// TwinCAT 3 PLC project Fraktal_Core
// Title: Fraktal_Core
// Company: fraktal-automation
// Author: fraktal-automation
// ProjectVersion: 0.1.0.5
// Description: Fraktal Core framework library: contracts, base classes (CM/EM/Unit), PermIntlk, profiler, connector base, recipe provider (Core 2.2).
// ProgramVersion: 3.1.4026.24
// libraries:
//   Tc2_Standard, * (Beckhoff Automation GmbH)
//   Tc2_EtherCAT, * (Beckhoff Automation GmbH)
//   Tc2_System, * (Beckhoff Automation GmbH)
//   Tc2_Utilities, * (Beckhoff Automation GmbH)
//   Tc3_Module, * (Beckhoff Automation GmbH)
// project tree:
//   BaseClasses/ FB_AccessManager.TcPOU, FB_AlarmLog.TcPOU, FB_AsciiDeviceCM.TcPOU, FB_ConfigPager.TcPOU, FB_ModuleBase.TcPOU, FB_ControlModuleBase.TcPOU (not stored), FB_CycleProfiler.TcPOU, FB_CompositeModuleBase.TcPOU, FB_EquipmentModuleBase.TcPOU (not stored), FB_SequenceBase.TcPOU (not stored), FB_UnitBase.TcPOU
//   Connectivity/ F_AppendTopologyConfig.TcPOU, FB_DeviceConnectorBase.TcPOU, FB_EcBusHealth.TcPOU, FB_EcFieldbusScanner.TcPOU (not stored), FB_IoTopologyPublisher.TcPOU, FB_LocalAccessProvider.TcPOU (not stored), FB_LocalPartCarrier.TcPOU (not stored), FB_LocalRecipeProvider.TcPOU (not stored), FB_LocalStationConfig.TcPOU, FB_SimByteChannel.TcPOU (not stored), FB_TcpChannelTc3.TcPOU (not stored)
//   DUTs/ E_AccessLevel.TcDUT (not stored), E_AlarmState.TcDUT (not stored), E_ByteChannelState.TcDUT (not stored), E_CarrierKind.TcDUT (not stored), E_Category.TcDUT (not stored), E_ChannelDir.TcDUT (not stored), E_ChannelKind.TcDUT (not stored), E_ExecState.TcDUT (not stored), E_FieldbusLossReaction.TcDUT (not stored), E_GatedAction.TcDUT (not stored), E_HbResult.TcDUT (not stored), E_LinkReaction.TcDUT (not stored), E_MachineState.TcDUT (not stored), E_Mode.TcDUT (not stored), E_ModeSwitchShield.TcDUT (not stored), E_PowerGroupKind.TcDUT (not stored), E_PowerState.TcDUT (not stored), E_SafetyDeviceKind.TcDUT (not stored), E_SafetyState.TcDUT (not stored), E_ModeSwitchStyle.TcDUT (not stored), E_ModuleType.TcDUT (not stored), E_NodeState.TcDUT (not stored), E_Reason.TcDUT (not stored), E_RecipeSource.TcDUT (not stored), E_ReleaseKind.TcDUT (not stored), E_ResetClass.TcDUT (not stored), E_RunStyle.TcDUT (not stored), E_Severity.TcDUT (not stored), E_StepResult.TcDUT (not stored), E_TimeClass.TcDUT (not stored), E_Verdict.TcDUT (not stored), ST_AccessPolicy.TcDUT (not stored), ST_AlarmEvent.TcDUT (not stored), ST_AlarmMeta.TcDUT (not stored), ST_BusNode.TcDUT (not stored), ST_CommandInfo.TcDUT (not stored), ST_CondRecord.TcDUT (not stored), ST_CycleProfile.TcDUT (not stored), ST_CycleSummary.TcDUT (not stored), ST_DecisionRequest.TcDUT (not stored), ST_Diagnostic.TcDUT (not stored), ST_FieldbusTopology.TcDUT (not stored), E_HmiRequestKind.TcDUT, ST_HmiRequest.TcDUT (not stored), ST_ConfigEntry.TcDUT, ST_ConfigPage.TcDUT, ST_HmiResponse.TcDUT (not stored), ST_IntlkCond.TcDUT (not stored), ST_IoChannel.TcDUT, ST_IoPointIdentity.TcDUT (not stored), ST_MeasRecord.TcDUT (not stored), ST_ModePolicy.TcDUT (not stored), ST_ModelField.TcDUT (not stored), ST_ModelId.TcDUT (not stored), ST_ModuleStatus.TcDUT (not stored), ST_ControlDomainStatus.TcDUT (not stored), ST_ControlPowerStatus.TcDUT (not stored), ST_PowerGroupStatus.TcDUT (not stored), ST_SafetyDeviceStatus.TcDUT (not stored), ST_SafetyStatus.TcDUT (not stored), ST_ModuleTiming.TcDUT (not stored), ST_Nameplate.TcDUT (not stored), ST_Oee.TcDUT (not stored), ST_OeeSample.TcDUT (not stored), ST_PartContext.TcDUT (not stored), ST_PartResult.TcDUT (not stored), ST_ReleaseReason.TcDUT (not stored), ST_ReleaseReport.TcDUT (not stored), ST_StepRecord.TcDUT, ST_StepTiming.TcDUT, ST_TimingRow.TcDUT (not stored), ST_UserRecord.TcDUT (not stored), ST_TcpVisionParCfg.TcDUT (not stored), ST_TcpVisionParCmd.TcDUT (not stored), ST_TcpVisionOutCmd.TcDUT (not stored), ST_TcpVisionOutImm.TcDUT (not stored), ST_TcpCodeReaderParCfg.TcDUT (not stored), ST_TcpCodeReaderParCmd.TcDUT (not stored), ST_TcpCodeReaderOutCmd.TcDUT (not stored), ST_TcpCodeReaderOutImm.TcDUT (not stored)
//   DeviceCMs/ FB_TcpCodeReaderCM.TcPOU, FB_TcpVisionCM.TcPOU (not stored)
//   Interfaces/ I_AccessProvider.TcIO (not stored), I_ByteChannel.TcIO (not stored), I_ControlModule.TcIO (not stored), I_DeviceConnector.TcIO (not stored), I_EquipmentModule.TcIO (not stored), I_EventSink.TcIO (not stored), I_FieldbusScanner.TcIO (not stored), I_ConfigSource.TcIO, I_Module.TcIO (not stored), I_PartCarrier.TcIO (not stored), I_SequenceHost.TcIO, I_RecipeProvider.TcIO (not stored), I_StationConfig.TcIO (not stored), I_Unit.TcIO (not stored), I_VerdictProvider.TcIO (not stored)
//   Params/ PL_Fraktal.TcGVL (not stored), PL_FraktalCompat.TcGVL (not stored), PL_TcpDevReasons.TcGVL (not stored)
//   PermIntlk/ FB_PermIntlk.TcPOU (not stored)
//   Platform/ F_Now.TcPOU (not stored), F_TimingUpdate.TcPOU (not stored)
// real-time tasks:
//   TASK PlcTask: cycle T#10ms, priority 20, ADS port 350
// I/O:
//   DEVICE =000+S-A610-A1 (EtherCAT), AmsNetId 0.0.0.0.2.1
//     =000+S-K010 (EK1200) [EK1200-5000 EtherCAT Power supply (2A E-Bus)]
//       =000+S-K010B1 (EL1809) [EL1809 16Ch. Dig. Input 24V, 3ms]
//       =000+S-K010C1 (EL2809) [EL2809 16Ch. Dig. Output 24V, 0.5A]
//       =000+S-K010D1 (EL6001) [EL6001 Interface (RS232)]
//       =000+S-K010E (EL9011) [EL9011 End Terminal]

// ---- DUTs/E_HmiRequestKind.TcDUT
// Core §3.10/§14 — generic OPC UA request mailbox operation.
// Append-only: ordinal values are a transport contract with every HMI adapter.
{attribute 'qualified_only'}
TYPE E_HmiRequestKind :
(
    NONE             := 0,
    LOGIN            := 1,
    LOGOUT           := 2,
    SET_MODE         := 3,
    SET_MODEL        := 4,
    START            := 5,
    STOP             := 6,
    CONTROL_ON       := 7,
    CONTROL_OFF      := 8,
    OPERATOR_RESET   := 9,
    DECISION_ANSWER  := 10,
    MANUAL_COMMAND   := 11,
    SET_RUN_STYLE    := 12,
    STEP_REQUEST     := 13,
    SET_HOLD_RUN     := 14,
    RELEASE_START    := 15,
    RELEASE_MANUAL   := 16,
    RELEASE_ACTION   := 17,
    RESET_OEE        := 18,
    WRITE_CONFIG     := 19,
    SHELVE_ALARM     := 20,
    UNSHELVE_ALARM   := 21,
    FORCE_CHANNEL    := 22,
    QUERY_CONFIG     := 23    // §3.10.2 config-manifest page request (IntValue = page)
) DINT;
END_TYPE

// ---- DUTs/ST_ConfigEntry.TcDUT
// Core §3.10.2 — one configuration value served through the request mailbox
// instead of the cyclic OPC UA tree. Scope selects the owner ('' = the root
// Unit itself, a qualified dotted module identity for a child, '#Fieldbus' for
// the bus topology). Item is the value's browse fragment in the server's array
// naming (e.g. 'Catalog/Catalog[2]/Label') so a generic HMI can rebuild the
// exact published path it would otherwise have read.
TYPE ST_ConfigEntry :
STRUCT
    Scope     : STRING(255);
    Item      : STRING(255);
    ValueText : STRING(255);   // typed by the HMI from the Item vocabulary
END_STRUCT
END_TYPE

// ---- DUTs/ST_ConfigPage.TcDUT
// Core §3.10.2 — one bounded page of the configuration manifest, published in
// ST_HmiResponse. The HMI requests QUERY_CONFIG with IntValue = PageIndex and
// walks 0..PageCount-1; Revision lets it detect a changed manifest (activation,
// changeover, config write) and refetch.
TYPE ST_ConfigPage :
STRUCT
    Revision   : UDINT;
    PageIndex  : INT;
    PageCount  : INT;
    EntryCount : INT;
    Entries    : ARRAY[1..PL_Fraktal.MAX_CONFIG_PAGE] OF ST_ConfigEntry;
END_STRUCT
END_TYPE

// ---- DUTs/ST_IoChannel.TcDUT
// Core §10.5.1 — one fieldbus I/O channel (published for the topology view §3.13)
TYPE ST_IoChannel :
STRUCT
    // §3.10.2 — tag/wiring identity is activation-static: excluded from the
    // cyclic OPC UA tree and served via the config manifest. Live I/O state
    // (values, force, quality, fault) stays cyclically published.
    {attribute 'OPC.UA.DA' := '0'}
    Name       : STRING(80);
    {attribute 'OPC.UA.DA' := '0'}
    DescriptionKey : STRING(160); // project/standard localization key
    {attribute 'OPC.UA.DA' := '0'}
    Address    : STRING(80);    // physical locator, e.g. EL1809 Ch5
    {attribute 'OPC.UA.DA' := '0'}
    Path       : STRING(255);   // unique channel path (force/audit identity)
    {attribute 'OPC.UA.DA' := '0'}
    ModulePath : STRING(255);   // owning module browse path for cross-navigation
    {attribute 'OPC.UA.DA' := '0'}
    Dir        : E_ChannelDir;
    {attribute 'OPC.UA.DA' := '0'}
    Kind       : E_ChannelKind;
    BoolValue  : BOOL;          // digital
    AnalogValue: REAL;          // analog (scaled)
    {attribute 'OPC.UA.DA' := '0'}
    Unit       : STRING(16);
    Forced     : BOOL;
    Quality    : BOOL;          // TRUE = good
    FaultActive: BOOL;          // a module diagnostic implicates this exact channel
    Diagnostic : STRING(255);   // localization key; Name remains the exact I/O tag
END_STRUCT
END_TYPE

// ---- DUTs/ST_StepRecord.TcDUT
// Core §6.5 — what the stall walk reads
TYPE ST_StepRecord :
STRUCT
    StepNo        : INT;
    StepName      : STRING(120);   // localization key
    AwaitingLabel : STRING(120);   // e.g. 'ClampStation.CLAMP' ('' if none)
    TimeClass     : E_TimeClass;   // Core §8.11.4(f) — WORK unless a genuine wait
    ExpectedTime  : TIME;          // defaults from the awaited command's timeout
    Conds         : ARRAY[1..PL_Fraktal.MAX_STEP_CONDS] OF ST_CondRecord;
END_STRUCT
END_TYPE

// ---- DUTs/ST_StepTiming.TcDUT
// Core §8.11.4(b)/(f) — one step of a cycle profile (Gantt/waterfall row)
TYPE ST_StepTiming :
STRUCT
    StepNo   : INT;
    StepName : STRING(120);   // localization key
    TimeClass    : E_TimeClass;  // WORK unless the step declared a wait class (§8.11.4(f))
    Started  : DT;           // synchronized wall clock (Core §2.7) — aligns across stations
    Duration : TIME;         // monotonic-clock duration (TC3 §8.11)
    Expected : TIME;         // §8.11.4(c) — the step's declared guard, drawn vs actual (0 = none)
END_STRUCT
END_TYPE

// ---- Interfaces/I_ConfigSource.TcIO
// Core §3.10.2 — a module that contributes entries to the root Unit's
// configuration manifest (static data deliberately excluded from the cyclic
// OPC UA tree and served through the QUERY_CONFIG mailbox instead).
// FB_ModuleBase implements it once for the base-owned facets; composites
// recurse their children, so a new module type inherits participation and
// only overrides M_AppendConfig to add type-owned static data (rare).
INTERFACE I_ConfigSource EXTENDS __System.IQueryInterface

// Append this module's (and its children's) manifest entries to the pager.
// Deterministic order across calls — the walk order defines the paging.
METHOD M_AppendConfig : BOOL
VAR_INPUT
    Pager : REFERENCE TO FB_ConfigPager;
END_VAR
END_METHOD

END_INTERFACE

// ---- Interfaces/I_SequenceHost.TcIO
// Core §6.7/§6.8 — the bridge from a separately-compiled sequence POU (SFC/ST/LD)
// to its owning module's protected framework services: step record, condition
// waits, run-style gate, part lifecycle, decisions, and completion/fault.
// FB_UnitBase implements it once; a sequence receives it at Setup. It carries
// framework plumbing ONLY — application decisions stay in the sequence's steps.
INTERFACE I_SequenceHost

// §6.11 publish a decision request
METHOD M_SequenceAskDecision
VAR_INPUT
    Req : ST_DecisionRequest;
END_VAR
END_METHOD

// §6.9(b) named plain-condition wait
METHOD M_SequenceAwait : BOOL
VAR_INPUT
    Idx : INT;
    Label : STRING(120);
    Ok : BOOL;
END_VAR
END_METHOD

// §6.11 withdraw an open request
METHOD M_SequenceClearDecision
END_METHOD

// §6.1 one-shot sequence completion (finite chains)
METHOD M_SequenceComplete
END_METHOD

// §8.11.2 carrier-less fallback counter
METHOD M_SequenceCountGood
END_METHOD

// §8.11.1 cycle-complete marker; FALSE = stop granted (chain must not loop)
METHOD M_SequenceEndOfCycle : BOOL
END_METHOD

// §6.9 first-out fault from a step
METHOD M_SequenceFault
VAR_INPUT
    Reason : E_Reason;
    DescriptionKey : STRING(255);
END_VAR
END_METHOD

// §3.16.3 EVENT_PART_PROCESSED (write-result-first; counts by verdict §8.11.2)
METHOD M_SequencePartProcessed : BOOL
VAR_INPUT
    Verdict : E_Verdict;
    Reason : E_Reason;
END_VAR
END_METHOD

// §3.16.3 EVENT_PART_RECEIVED
METHOD M_SequencePartReceived : BOOL
END_METHOD

// §3.16.1 measured value
METHOD M_SequencePartRecord : BOOL
VAR_INPUT
    RecordName : STRING(64);
    Value : LREAL;
    Minimum : LREAL;
    Maximum : LREAL;
    Target : LREAL;
    EngUnit : STRING(16);
END_VAR
END_METHOD

// §3.16.3 EVENT_PART_PROCESSING_STARTED
METHOD M_SequencePartStarted
END_METHOD

// §6.5 step record (feeds the §6.9 walk and the §8.11.4 profiler)
METHOD M_SequenceSetStep
VAR_INPUT
    StepNo : INT;
    StepName : STRING(120);
    Awaits : I_Module;
    AwaitingLabel : STRING(120);
    TimeClass : E_TimeClass;
    ExpectedTime : TIME;
END_VAR
END_METHOD

// §3.4.2 run-style pacing gate
METHOD M_SequenceStepGate : BOOL
VAR_INPUT
    Steppable : BOOL;
END_VAR
END_METHOD

// §3.4/§8.11 — accept a pending Stop BETWEEN cycles: abandon the open cycle
// profile (no §8.11.1 cycle is counted for a wait-only fragment) and complete.
METHOD M_SequenceStopNow
END_METHOD

// §3.4 — TRUE while a Stop is requested and the sequence still runs. A chain
// polls this at its between-cycles wait so a stop need not ride out a phantom cycle.
METHOD M_SequenceStopPending : BOOL
END_METHOD

// §6.11 consume the answer once (0 = none yet)
METHOD M_SequenceTakeDecision : INT
END_METHOD

END_INTERFACE

// ---- BaseClasses/FB_AccessManager.TcPOU
// Core §7.7(c) — per-root session + enforcement. Login/logout is DATA-DRIVEN
// (§3.10(a')): the HMI writes ReqUser/ReqSecret and pulses ReqLogin/ReqLogout;
// the secret is cleared after every attempt. Policy default: fully open (§7.7(b)).
FUNCTION_BLOCK FB_AccessManager
VAR_INPUT
    ReqUser   : STRING(32);          // HMI-writable login request
    ReqSecret : STRING(32);          // cleared after each attempt (§7.7(c))
    ReqLogin  : BOOL;
    ReqLogout : BOOL;
END_VAR
VAR_OUTPUT
    CurrentUser  : STRING(32);
    CurrentLevel : E_AccessLevel;    // HMI greys controls from this; PLC re-checks
    LoginFailed  : BOOL;             // last attempt outcome (HMI feedback)
END_VAR
VAR PERSISTENT
    Policy : ST_AccessPolicy;        // §3.8a station config; edit gated by ACCESS_POLICY
END_VAR
VAR
    {attribute 'OPC.UA.DA' := '0'}
    _provider : I_AccessProvider;
    {attribute 'OPC.UA.DA' := '0'}
    _log      : POINTER TO FB_AlarmLog;
    _tIdle    : TON;
END_VAR

// event/session handling is in Cyclic (called by the owning Unit each scan)

METHOD Cyclic : BOOL
VAR
    lvl : E_AccessLevel;
    loginHandled : BOOL;
    logoutHandled : BOOL;
END_VAR
loginHandled := ReqLogin;
IF loginHandled THEN
    ReqLogin := FALSE;
    lvl := E_AccessLevel.NONE;
    IF _provider <> 0 THEN
        lvl := _provider.Authenticate(User := ReqUser, Secret := ReqSecret);
    END_IF
    ReqSecret := '';                                   // never retain the secret
    IF lvl > E_AccessLevel.NONE THEN
        CurrentUser := ReqUser;
        CurrentLevel := lvl;
        LoginFailed := FALSE;
        _M_Audit('std.audit.login', CurrentUser);
    ELSE
        LoginFailed := TRUE;
        _M_Audit('std.audit.loginFailed', ReqUser);
    END_IF
END_IF
logoutHandled := ReqLogout;
IF logoutHandled THEN
    ReqLogout := FALSE;
    IF CurrentLevel > E_AccessLevel.NONE THEN
        _M_Audit('std.audit.logout', CurrentUser);
        CurrentUser := '';
        CurrentLevel := E_AccessLevel.NONE;
    END_IF
END_IF
// idle auto-logout (§7.7(c)); any successful login rearms it
_tIdle(IN := (Policy.SessionTimeout > T#0S) AND (CurrentLevel > E_AccessLevel.NONE) AND NOT loginHandled,
       PT := Policy.SessionTimeout);
IF _tIdle.Q THEN
    _M_Audit('std.audit.autoLogout', CurrentUser);
    CurrentUser := '';
    CurrentLevel := E_AccessLevel.NONE;
END_IF
Cyclic := TRUE;
END_METHOD

// Startup/station-configuration seam; runtime HMI writes remain Unit-gated.
METHOD ConfigureRequired : BOOL
VAR_INPUT
    Gate : E_GatedAction;
    Level : E_AccessLevel;
END_VAR
IF (TO_INT(Gate) < 0) OR (TO_INT(Gate) > TO_INT(E_GatedAction.POWER_CONTROL)) THEN
    ConfigureRequired := FALSE;
ELSE
    Policy.Required[TO_INT(Gate)] := Level;
    ConfigureRequired := TRUE;
END_IF
END_METHOD

// ST-facing request seam. OPC UA clients continue to write the published request data.
METHOD RequestLogin : BOOL
VAR_INPUT
    User : STRING(32);
    Secret : STRING(32);
END_VAR
ReqUser := User;
ReqSecret := Secret;
ReqLogin := TRUE;
RequestLogin := TRUE;
END_METHOD

// ST-facing request seam; the cyclic edge handler performs the state change and audit.
METHOD RequestLogout : BOOL
ReqLogout := TRUE;
RequestLogout := TRUE;
END_METHOD

// pure check for UI/logic — no logging
METHOD Permits : BOOL
VAR_INPUT
    Gate : E_GatedAction;
END_VAR
Permits := TO_DINT(CurrentLevel) >= TO_DINT(Policy.Required[TO_INT(Gate)]);
END_METHOD

// gated-entry check: a DENIED attempt is audited as a MESSAGE event (§8.3/§7.7(c))
METHOD PermitsLogged : BOOL
VAR_INPUT
    Gate : E_GatedAction;
END_VAR
PermitsLogged := Permits(Gate := Gate);
IF NOT PermitsLogged THEN
    _M_Audit('std.audit.accessDenied', CurrentUser);
END_IF
END_METHOD

METHOD Setup : BOOL
VAR_INPUT
    Provider : I_AccessProvider;
    pAlarmLog : POINTER TO FB_AlarmLog;
END_VAR
IF Provider <> 0 THEN
    _provider := Provider;                  // Unit OnInit may attach only the audit log
END_IF
_log := pAlarmLog;
Setup := TRUE;
END_METHOD

// audit trail for free: come+gone MESSAGE lands in the §8.3 ring
METHOD PRIVATE _M_Audit
VAR_INPUT
    What : STRING(64);
    Who : STRING(32);
END_VAR
VAR
    auditSlot : INT;
    txt : STRING(255);
END_VAR
IF _log = 0 THEN
    RETURN;
END_IF
txt := CONCAT(What, ': ');
txt := CONCAT(txt, Who);
auditSlot := _log^.Raise(Reason := E_Reason.NONE, Text := txt,
                 Source := 'Access', Severity := E_Severity.LOW,
                 Category := E_Category.SYSTEM, ResetClass := E_ResetClass.AUTO_RESET);
IF auditSlot > 0 THEN
    _log^.Gone(Slot := auditSlot);                     // instant come+gone -> ring entry
END_IF
END_METHOD

END_FUNCTION_BLOCK

// ---- BaseClasses/FB_AlarmLog.TcPOU
// Core §8.3 — per-Unit alarm & event log: active list + closed ring, durations,
// AUTO/MANUAL reset classes, optional historian sink. Fixed-size, never allocates.
FUNCTION_BLOCK FB_AlarmLog
VAR_OUTPUT
    Active    : ARRAY[1..PL_Fraktal.MAX_ALARM_ACTIVE] OF ST_AlarmEvent;  // ACTIVE/WAIT_RESET
    NActive   : INT;
    Ring      : ARRAY[1..PL_Fraktal.MAX_ALARM_RING] OF ST_AlarmEvent;    // closed, newest at RingHead
    RingHead  : INT;
    Blocking  : BOOL;    // any MANUAL_RESET event ACTIVE/WAIT_RESET (§8.3(b))
    Truncated : BOOL;
    // §3.10.2 — rationalization records are static config; excluded from the
    // cyclic OPC UA tree (served via the manifest when an HMI needs them).
    {attribute 'OPC.UA.DA' := '0'}
    Meta      : ARRAY[1..PL_Fraktal.MAX_ALARM_META] OF ST_AlarmMeta;  // §8.9 rationalization
    {attribute 'OPC.UA.DA' := '0'}
    MetaCount : INT;
END_VAR
VAR
    {attribute 'OPC.UA.DA' := '0'}
    _sink    : I_EventSink;
    _comeMs  : ARRAY[1..PL_Fraktal.MAX_ALARM_ACTIVE] OF DWORD;   // monotonic (TC3 §8.11)
    _shelfMs : ARRAY[1..PL_Fraktal.MAX_ALARM_ACTIVE] OF UDINT;   // §8.10 countdown (0 = not shelved)
    _cycLast : TIME;                                             // Cyclic delta stamp
END_VAR

// event-driven; no cyclic body

// §8.3(c) — open a non-channel-specific event; returns slot (0 = full).
METHOD Raise : INT
VAR_INPUT
    Reason : E_Reason;
    Text : STRING(255);
    Source : STRING(255);
    Severity : E_Severity;
    Category : E_Category;
    ResetClass : E_ResetClass;
END_VAR
Raise := _M_Raise(Reason := Reason, Text := Text, Source := Source,
    IoTag := '', IoAddress := '', Severity := Severity, Category := Category,
    ResetClass := ResetClass);
END_METHOD

// §8.3(c) — open an event; returns its slot id (0 = table full -> Truncated)
METHOD PRIVATE _M_Raise : INT
VAR_INPUT
    Reason : E_Reason;
    Text : STRING(255);
    Source : STRING(255);
    IoTag : STRING(80);
    IoAddress : STRING(80);
    Severity : E_Severity;
    Category : E_Category;
    ResetClass : E_ResetClass;
END_VAR
VAR
    i, slot : INT;
END_VAR
slot := 0;
FOR i := 1 TO PL_Fraktal.MAX_ALARM_ACTIVE DO
    IF Active[i].State = E_AlarmState.CLOSED THEN
        slot := i;
        EXIT;
    END_IF
END_FOR
IF slot = 0 THEN
    Truncated := TRUE;
    _M_Raise := 0;
    RETURN;
END_IF
Active[slot].ReasonCode  := Reason;
Active[slot].Description := Text;
Active[slot].SourcePath  := Source;
Active[slot].IoTag       := IoTag;
Active[slot].IoAddress   := IoAddress;
Active[slot].Severity    := Severity;
Active[slot].Category    := Category;
Active[slot].ResetClass  := ResetClass;
Active[slot].State       := E_AlarmState.ACTIVE;
Active[slot].ComeAt      := F_Now();
Active[slot].GoneAt      := DT#1970-01-01-00:00:00;
Active[slot].ResetAt     := DT#1970-01-01-00:00:00;
Active[slot].Duration    := T#0S;
Active[slot].Shelved     := FALSE;
Active[slot].ShelvedUntil:= DT#1970-01-01-00:00:00;
_shelfMs[slot] := 0;
_comeMs[slot] := TIME_TO_DWORD(TIME());
NActive := NActive + 1;
_M_UpdateBlocking();
IF _sink <> 0 THEN
    _sink.OnEvent(Ev := Active[slot]);              // come notification (§8.3(d))
END_IF
_M_Raise := slot;
END_METHOD

// §8.3(c) — open an ERROR event straight from a first-out diagnostic (no re-authoring)
METHOD RaiseDiag : INT
VAR_INPUT
    D : ST_Diagnostic;
    ResetClass : E_ResetClass;
END_VAR
RaiseDiag := _M_Raise(Reason := D.ReasonCode, Text := D.Description,
                   Source := D.SourcePath, IoTag := D.IoTag, IoAddress := D.IoAddress,
                   Severity := D.Severity, Category := D.Category,
                   ResetClass := ResetClass);
END_METHOD

// §8.3(b) — condition re-established: AUTO_RESET closes with Duration;
// MANUAL_RESET stays blocking in WAIT_RESET until OperatorReset.
METHOD Gone : BOOL
VAR_INPUT
    Slot : INT;
END_VAR
Gone := FALSE;
IF (Slot < 1) OR (Slot > PL_Fraktal.MAX_ALARM_ACTIVE) THEN
    RETURN;
END_IF
IF Active[Slot].State <> E_AlarmState.ACTIVE THEN
    RETURN;
END_IF
Active[Slot].GoneAt   := F_Now();
Active[Slot].Duration := DWORD_TO_TIME(TIME_TO_DWORD(TIME()) - _comeMs[Slot]);   // wrap-safe
IF Active[Slot].ResetClass = E_ResetClass.AUTO_RESET THEN
    _M_Close(Slot);
ELSE
    Active[Slot].State := E_AlarmState.WAIT_RESET;   // still blocking (§8.3(b))
END_IF
Gone := TRUE;
END_METHOD

// §8.3(b) — deliberate, release-gated operator action (§7.6/§14): closes
// MANUAL_RESET events whose condition is gone. NEVER self-invoked (§9.3 principle).
METHOD OperatorReset : BOOL
VAR
    i : INT;
END_VAR
OperatorReset := FALSE;
FOR i := 1 TO PL_Fraktal.MAX_ALARM_ACTIVE DO
    IF Active[i].State = E_AlarmState.WAIT_RESET THEN
        Active[i].ResetAt := F_Now();
        _M_Close(i);
        OperatorReset := TRUE;
    END_IF
END_FOR
END_METHOD

METHOD SetSink : BOOL
VAR_INPUT
    Sink : I_EventSink;
END_VAR
_sink := Sink;
SetSink := TRUE;
END_METHOD

METHOD PRIVATE _M_Close
VAR_INPUT
    Slot : INT;
END_VAR
Active[Slot].State := E_AlarmState.CLOSED;
RingHead := (RingHead MOD PL_Fraktal.MAX_ALARM_RING) + 1;
Ring[RingHead] := Active[Slot];
Ring[RingHead].State := E_AlarmState.CLOSED;
NActive := NActive - 1;
_M_UpdateBlocking();
IF _sink <> 0 THEN
    _sink.OnEvent(Ev := Ring[RingHead]);            // close notification with Duration (§8.3(d))
END_IF
END_METHOD

METHOD PRIVATE _M_UpdateBlocking
VAR
    i : INT;
    b : BOOL;
END_VAR
b := FALSE;
FOR i := 1 TO PL_Fraktal.MAX_ALARM_ACTIVE DO
    IF (Active[i].ResetClass = E_ResetClass.MANUAL_RESET)
    AND (Active[i].State <> E_AlarmState.CLOSED) THEN
        b := TRUE;
        EXIT;
    END_IF
END_FOR
Blocking := b;
END_METHOD

// §8.9 — register/update the rationalization record for a ReasonCode (idempotent).
// Modules/Units call at Setup. No record => the reason is NOT shelvable (§8.10).
METHOD RegisterMeta : BOOL
VAR_INPUT
    Reason         : E_Reason;
    OperatorAction : STRING(255);
    Consequence    : STRING(255);
    Shelvable      : BOOL;
END_VAR
VAR
    i : INT;
END_VAR
FOR i := 1 TO MetaCount DO
    IF Meta[i].ReasonCode = Reason THEN
        Meta[i].OperatorAction := OperatorAction;
        Meta[i].Consequence := Consequence;
        Meta[i].Shelvable := Shelvable;
        RegisterMeta := TRUE;
        RETURN;
    END_IF
END_FOR
IF MetaCount >= PL_Fraktal.MAX_ALARM_META THEN
    RegisterMeta := FALSE;
    RETURN;
END_IF
MetaCount := MetaCount + 1;
Meta[MetaCount].ReasonCode := Reason;
Meta[MetaCount].OperatorAction := OperatorAction;
Meta[MetaCount].Consequence := Consequence;
Meta[MetaCount].Shelvable := Shelvable;
RegisterMeta := TRUE;
END_METHOD

// §8.10 — may this active slot be shelved? SAFETY never; no meta record => no.
METHOD PROTECTED _M_Shelvable : BOOL
VAR_INPUT
    Slot : INT;
END_VAR
VAR
    i : INT;
END_VAR
_M_Shelvable := FALSE;
IF Slot < 1 OR Slot > PL_Fraktal.MAX_ALARM_ACTIVE THEN
    RETURN;
END_IF
IF Active[Slot].State = E_AlarmState.CLOSED THEN
    RETURN;
END_IF
IF Active[Slot].Category = E_Category.SAFETY THEN
    RETURN;                              // §8.10: safety never shelvable
END_IF
FOR i := 1 TO MetaCount DO
    IF Meta[i].ReasonCode = Active[Slot].ReasonCode THEN
        _M_Shelvable := Meta[i].Shelvable;
        RETURN;
    END_IF
END_FOR
// no rationalization record => not shelvable (rationalize first, §8.10)
END_METHOD

// §8.10 — suppress ANNUNCIATION of an active alarm for DurationS seconds (capped).
// Control is untouched: Blocking, interlocks, release reports all still see it.
// Caller has already checked §7.7 ALARM_SHELVE; the shelf itself is logged here.
METHOD Shelve : BOOL
VAR_INPUT
    Slot      : INT;
    DurationS : UDINT;
END_VAR
VAR
    auditSlot : INT;
END_VAR
IF NOT _M_Shelvable(Slot := Slot) THEN
    Shelve := FALSE;
    RETURN;
END_IF
IF DurationS = 0 THEN
    Shelve := FALSE;                              // every shelf is time-bounded
    RETURN;
END_IF
IF DurationS > PL_Fraktal.MAX_SHELF_S THEN
    DurationS := PL_Fraktal.MAX_SHELF_S;         // §8.10 time-bounded
END_IF
Active[Slot].Shelved := TRUE;
Active[Slot].ShelvedUntil := DWORD_TO_DT(DT_TO_DWORD(F_Now()) + DurationS);
_shelfMs[Slot] := DurationS * 1000;
auditSlot := Raise(Reason := E_Reason.NONE,
    Text := 'std.audit.alarmShelved', Source := Active[Slot].SourcePath,
    Severity := E_Severity.LOW, Category := E_Category.SYSTEM, ResetClass := E_ResetClass.AUTO_RESET);
IF auditSlot > 0 THEN Gone(Slot := auditSlot); END_IF
Shelve := TRUE;
END_METHOD

// §8.10 — restore annunciation (operator or auto-expiry). Logged.
METHOD Unshelve : BOOL
VAR_INPUT
    Slot : INT;
END_VAR
VAR
    auditSlot : INT;
END_VAR
IF Slot < 1 OR Slot > PL_Fraktal.MAX_ALARM_ACTIVE THEN
    Unshelve := FALSE;
    RETURN;
END_IF
IF NOT Active[Slot].Shelved THEN
    Unshelve := FALSE;
    RETURN;
END_IF
Active[Slot].Shelved := FALSE;
_shelfMs[Slot] := 0;
auditSlot := Raise(Reason := E_Reason.NONE,
    Text := 'std.audit.alarmUnshelved', Source := Active[Slot].SourcePath,
    Severity := E_Severity.LOW, Category := E_Category.SYSTEM, ResetClass := E_ResetClass.AUTO_RESET);
IF auditSlot > 0 THEN Gone(Slot := auditSlot); END_IF
Unshelve := TRUE;
END_METHOD

// §8.10 — auto-unshelve countdown (owning Unit ticks this each scan).
METHOD Cyclic : BOOL
VAR
    currentTime : TIME;
    deltaMs     : UDINT;
    i   : INT;
END_VAR
currentTime := TIME();                 // monotonic duration clock
IF _cycLast = T#0S THEN
    _cycLast := currentTime;
    Cyclic := TRUE;
    RETURN;
END_IF
deltaMs := TIME_TO_UDINT(currentTime) - TIME_TO_UDINT(_cycLast);
_cycLast := currentTime;
FOR i := 1 TO PL_Fraktal.MAX_ALARM_ACTIVE DO
    IF Active[i].Shelved AND _shelfMs[i] > 0 THEN
        IF _shelfMs[i] > deltaMs THEN
            _shelfMs[i] := _shelfMs[i] - deltaMs;
        ELSE
            _shelfMs[i] := 0;
            Unshelve(Slot := i);                 // §8.10 auto-expire (logged by Unshelve)
        END_IF
    END_IF
END_FOR
Cyclic := TRUE;
END_METHOD

END_FUNCTION_BLOCK

// ---- BaseClasses/FB_AsciiDeviceCM.TcPOU
// Core §3.15.1a — CM base for ASCII request/response devices over I_ByteChannel
// (vision sensors, code readers, gauges). One-outstanding-request state machine:
// SendRequest -> await terminated response -> _M_OnResponse hook; silence -> fault
// 10402. Written ONCE against the neutral seam: porting = swap the channel (O4/O8).
// Reconnect: bounded retry via the channel; link state published for Annex D facet.
FUNCTION_BLOCK ABSTRACT FB_AsciiDeviceCM EXTENDS FB_ControlModuleBase
VAR
    Host        : STRING(80);          // §3.8 config (per deployment)
    Port        : UINT;
    Terminator  : STRING(2) := '$R';   // CR default; device profile may override
    RespTimeout : TIME := T#2S;
    LinkState   : E_ByteChannelState;  // published (Annex D link facet)
    LastResponse: STRING(255);         // published (diagnosis)
END_VAR
VAR
    {attribute 'OPC.UA.DA' := '0'}
    _chan     : I_ByteChannel;
    _rx       : STRING(255);
    _pending  : BOOL;                  // one outstanding request
    _tResp    : TON;
    _tRetry   : TON;
    _retryMs  : TIME := T#500MS;       // bounded backoff (doubles to 10s)
    _openTried : BOOL;                 // backoff spaces RE-tries; the first Open is immediate
END_VAR

;  // driven via Cyclic (base) -> OnCyclic below

// wire the transport + endpoint. Call from the profile's Setup after _M_SetName.
METHOD SetupDevice : BOOL
VAR_INPUT
    Chan : I_ByteChannel;
    DevHost : STRING(80);
    DevPort : UINT;
END_VAR
IF Chan = 0 OR DevHost = '' THEN
    _M_FaultN(PL_TcpDevReasons.DEV_CFG_INVALID, 'std.error.deviceConnectionNotConfigured');
    SetupDevice := FALSE;
    RETURN;
END_IF
_chan := Chan;
Host := DevHost;
Port := DevPort;
SetupDevice := TRUE;
END_METHOD

// channel management + RX framing. Profiles override _M_OnResponse, not this.
METHOD PROTECTED OnCyclic : DINT
VAR
    pos : INT;
    resp : STRING(255);
END_VAR
OnCyclic := SUPER^.OnCyclic();
IF _chan = 0 THEN
    RETURN;
END_IF
_chan.Tick();
LinkState := _chan.State();
CASE LinkState OF
    E_ByteChannelState.CLOSED:
        IF NOT _openTried THEN
            _openTried := TRUE;                    // first sight of CLOSED: connect NOW
            _chan.Open(Host := Host, Port := Port);
            LinkState := _chan.State();            // a synchronous transport is OPEN this scan
        ELSE
            _tRetry(IN := TRUE, PT := _retryMs);   // failed before: bounded backoff (§3.15.2 spirit)
            IF _tRetry.Q THEN
                _tRetry(IN := FALSE);
                _chan.Open(Host := Host, Port := Port);
                LinkState := _chan.State();
                IF _retryMs < T#10S THEN
                    _retryMs := _retryMs * 2;
                END_IF
            END_IF
        END_IF
    E_ByteChannelState.OPEN:
        _openTried := FALSE;
        _retryMs := T#500MS;
        _chan.Poll(Buffer := _rx);
        pos := FIND(_rx, Terminator);
        IF pos > 0 THEN
            resp := LEFT(_rx, pos - 1);
            _rx := DELETE(_rx, pos + LEN(Terminator) - 1, 1);
            _pending := FALSE;
            _tResp(IN := FALSE);
            LastResponse := resp;
            _M_OnResponse(Response := resp);
        ELSIF LEN(_rx) >= 250 THEN
            _rx := '';
            _M_FaultN(PL_TcpDevReasons.DEV_RX_OVERFLOW, 'std.error.deviceResponseOverflow');
        END_IF
    E_ByteChannelState.FAULT:
        IF _pending THEN
            _pending := FALSE;
            _tResp(IN := FALSE);
        END_IF
        _M_FaultN(PL_TcpDevReasons.DEV_CHANNEL_FAULT, 'std.error.transportChannelFault');
        _chan.Close();
ELSE
    _M_FaultN(PL_TcpDevReasons.DEV_CHANNEL_FAULT, 'std.error.byteChannelStateInvalid');
    _chan.Close();
END_CASE
// response timeout watch
_tResp(IN := _pending, PT := RespTimeout);
IF _tResp.Q THEN
    _pending := FALSE;
    _tResp(IN := FALSE);
    _M_FaultN(PL_TcpDevReasons.DEV_RESP_TIMEOUT, 'std.error.deviceResponseTimeout');
END_IF
END_METHOD

// issue one request (terminator appended). FALSE if not connected or one pending.
METHOD SendRequest : BOOL
VAR_INPUT
    Text : STRING(250);
END_VAR
// live channel state: the cached LinkState is one scan old and would reject a
// request issued in the same scan the transport opened.
IF _chan = 0 OR (_chan.State() <> E_ByteChannelState.OPEN) THEN
    _M_FaultN(PL_TcpDevReasons.DEV_NOT_CONNECTED, 'std.error.deviceNotConnected');
    SendRequest := FALSE;
    RETURN;
END_IF
IF _pending THEN
    SendRequest := FALSE;              // one-outstanding-request contract
    RETURN;
END_IF
_pending := _chan.Send(Text := CONCAT(Text, Terminator));
SendRequest := _pending;
END_METHOD

// profile hook: parse one terminated response. Raise DEV_PROTOCOL on garbage.
METHOD PROTECTED _M_OnResponse
VAR_INPUT
    Response : STRING(255);
END_VAR
;
END_METHOD

END_FUNCTION_BLOCK

// ---- BaseClasses/FB_ConfigPager.TcPOU
// Core §3.10.2 — windowed writer for the configuration manifest. QUERY_CONFIG
// re-walks the whole export enumeration each request; the pager counts every
// appended entry and stores only the requested page window into the published
// ST_ConfigPage, so no full manifest buffer ever exists in PLC memory and the
// walk order alone defines the paging. Exporters call M_Append*/ignore paging.
FUNCTION_BLOCK FB_ConfigPager
VAR
    {attribute 'OPC.UA.DA' := '0'}
    _pTarget : POINTER TO ST_ConfigPage;
    _cursor  : DINT;   // entries appended so far in this walk
    _first   : DINT;   // first cursor index stored in the window (0-based)
END_VAR

; // stateless between requests — driven entirely by M_Setup/M_Append/M_Finish

// Begin one QUERY_CONFIG walk targeting the published page window.
METHOD M_Setup : BOOL
VAR_INPUT
    Target    : POINTER TO ST_ConfigPage;
    PageIndex : INT;
    Revision  : UDINT;
END_VAR
M_Setup := FALSE;
IF Target = 0 THEN
    RETURN;
END_IF
_pTarget := Target;
_cursor := 0;
IF PageIndex < 0 THEN
    _first := 0;
ELSE
    _first := TO_DINT(PageIndex) * TO_DINT(PL_Fraktal.MAX_CONFIG_PAGE);
END_IF
_pTarget^.Revision := Revision;
_pTarget^.PageIndex := SEL(PageIndex < 0, PageIndex, 0);
_pTarget^.PageCount := 0;
_pTarget^.EntryCount := 0;
M_Setup := TRUE;
END_METHOD

// Append one manifest entry; stored only when it falls inside the page window.
// Always returns TRUE so exporters can chain without branching.
METHOD M_Append : BOOL
VAR_INPUT
    Scope     : STRING(255);
    Item      : STRING(255);
    ValueText : STRING(255);
END_VAR
VAR
    slot : DINT;
END_VAR
M_Append := TRUE;
IF _pTarget = 0 THEN
    RETURN;
END_IF
slot := _cursor - _first;   // window-relative 0-based position
_cursor := _cursor + 1;
IF (slot < 0) OR (slot >= TO_DINT(PL_Fraktal.MAX_CONFIG_PAGE)) THEN
    RETURN;                 // outside the requested window — counted, not stored
END_IF
_pTarget^.Entries[TO_INT(slot) + 1].Scope := Scope;
_pTarget^.Entries[TO_INT(slot) + 1].Item := Item;
_pTarget^.Entries[TO_INT(slot) + 1].ValueText := ValueText;
_pTarget^.EntryCount := TO_INT(slot) + 1;
END_METHOD

METHOD M_AppendNumber : BOOL
VAR_INPUT
    Scope  : STRING(255);
    Item   : STRING(255);
    Number : DINT;
END_VAR
M_AppendNumber := M_Append(Scope := Scope, Item := Item,
    ValueText := TO_STRING(Number));
END_METHOD

// Close the walk: publish the total page count for the HMI's fetch loop.
METHOD M_Finish : BOOL
M_Finish := FALSE;
IF _pTarget = 0 THEN
    RETURN;
END_IF
_pTarget^.PageCount := TO_INT(
    (_cursor + TO_DINT(PL_Fraktal.MAX_CONFIG_PAGE) - 1)
    / TO_DINT(PL_Fraktal.MAX_CONFIG_PAGE));
M_Finish := TRUE;
END_METHOD

END_FUNCTION_BLOCK

// ---- BaseClasses/FB_ModuleBase.TcPOU
// Core §2.2 / §6.1 — the PLCopen lifecycle written ONCE (template method).
// A concrete type EXTENDS this base, declares its Command/HAL/ParCfg members, and
// overrides only _M_Dispatch (+ optionally hooks and recipe transaction methods).
// Edge handling, ExecState mapping, Execute-drop reset, ErrorID publication, and
// abort routing are inherited. Conformance rows T1/T4 (Core §5.7) are satisfied here
// and proven once in FB_Base_Tests.
FUNCTION_BLOCK ABSTRACT FB_ModuleBase IMPLEMENTS I_Module, I_ConfigSource
VAR_INPUT
    Execute : BOOL;    // rising edge starts the command (Core §6.1)
    Abort   : BOOL;    // requests a controlled abort
END_VAR
VAR_OUTPUT
    Busy    : BOOL;
    Done    : BOOL;
    Error   : BOOL;
    Aborted : BOOL;
    ErrorID : DWORD;   // = TO_DWORD(first-out ReasonCode), Core §8.8
END_VAR
VAR_OUTPUT
    Status : ST_ModuleStatus;   // Core §3.10(a')/§6.9(a) — the OPC UA data mirror
    Timing : ST_ModuleTiming;   // Core §8.11.4(a) — per-command timing, captured here once
    // §3.10.2 — static facets stay OFF the cyclic OPC UA tree and are served
    // through the QUERY_CONFIG manifest instead (M_AppendConfig).
    {attribute 'OPC.UA.DA' := '0'}
    Nameplate   : ST_Nameplate;  // §3.10.1 asset identity (set at Setup; empty = none)
    {attribute 'OPC.UA.DA' := '0'}
    Catalog     : ARRAY[1..PL_Fraktal.MAX_CMD_CATALOG] OF ST_CommandInfo;  // §7.6.1 published command list
    {attribute 'OPC.UA.DA' := '0'}
    CatalogCount: INT;
    Safety       : ST_SafetyStatus;       // §9 optional read-only safety facet (Present=FALSE if absent)
    ControlPower : ST_ControlPowerStatus; // §9 optional control/power facet
END_VAR
VAR
    _name  : STRING(80);
    _exec  : E_ExecState := E_ExecState.READY;
    _step  : INT;
    _diag  : ST_Diagnostic;
    _rTrig : R_TRIG;
    _abortErrTrig : R_TRIG;
    _initialized : BOOL;
    _prevExec   : E_ExecState;
    _manualCmd  : DINT;          // §7.6.1 pending manual command value (0 = none)
    _manualReq  : BOOL;
    _manualActive : BOOL;        // one-shot manual request owns Execute until terminal state
    _cmdArmed   : BOOL;          // terminal state came from a command; gates the §6.1 reset
    _cmdId      : DINT;          // set by _M_TagCommand (one line per type, §8.11.4(a))
    _cmdLabel   : STRING(120);
    _tCmdStart  : DWORD;         // monotonic ms at command start (TC3 §8.11)
END_VAR

// FB body just runs the lifecycle; parents may call the instance or Cyclic() (I_Module)
Cyclic();

// Core §6.1 — edge -> hooks -> dispatch -> map -> Execute-drop reset
METHOD Cyclic : BOOL
VAR
    commandStarted : BOOL;
END_VAR
commandStarted := FALSE;
// Execute-drop reset (Core §6.1): a COMMAND-produced terminal state published in
// an earlier scan plus Execute low resets to READY BEFORE this scan's mapping, so
// the outputs go idle in the same call. A completion later this scan still maps
// its one-cycle DONE/ERROR/ABORTED pulse first (PLCopen). Faults raised OUTSIDE a
// command (recipe/config at Setup, cyclic condition monitors) latch (§3.8/§8.3):
// Execute was never high, so the handshake reset does not consume them.
IF (NOT Execute) AND _cmdArmed
AND ((_exec = E_ExecState.DONE) OR (_exec = E_ExecState.ERROR) OR (_exec = E_ExecState.ABORTED)) THEN
    _exec := E_ExecState.READY;
    _cmdArmed := FALSE;
END_IF

_rTrig(CLK := Execute);
// A fresh command edge may also RETRY from a latched non-command fault: the edge
// clears the diagnostic and re-runs validation, which re-faults if the cause remains.
IF _rTrig.Q AND ((_exec = E_ExecState.READY)
    OR ((_exec = E_ExecState.ERROR) AND NOT _cmdArmed)) THEN
    _exec := E_ExecState.BUSY;      // ParCmd of the concrete type is latched on this edge
    _cmdArmed := TRUE;
    _step := 10;
    _M_ClearDiag();
    _tCmdStart := TIME_TO_DWORD(TIME());          // §8.11.4(a) command-timing start
    commandStarted := TRUE;
END_IF

IF NOT _initialized THEN
    _initialized := TRUE;
    OnInit();                        // Core §3.14 one-shot for every module tier
END_IF
IF commandStarted THEN
    OnCommandStart();                // one-shot after init, before cyclic/dispatch
END_IF
OnCyclic();                          // Core §3.14 hook: background management, no outputs

IF Abort AND (_exec = E_ExecState.BUSY) THEN
    OnAbort();                       // Core §3.14 hook: device-safe abort action
END_IF
_abortErrTrig(CLK := Abort AND (_exec = E_ExecState.ERROR));
IF _abortErrTrig.Q THEN
    OnAbortInError();                // distinct recovery hook; ERROR remains latched
END_IF

IF _exec = E_ExecState.BUSY THEN
    _M_Dispatch();                   // the ONLY thing a type must write (Core §2.2)
END_IF

// §8.11.4(a) — close the command's timing row on leaving BUSY (DONE/ERROR/ABORTED)
IF (_prevExec = E_ExecState.BUSY) AND (_exec <> E_ExecState.BUSY) THEN
    _M_RecordCmdTiming(TIME_TO_DWORD(TIME()) - _tCmdStart);   // wrap-safe diff (TC3 §8.11)
END_IF
_prevExec := _exec;

Busy    := (_exec = E_ExecState.BUSY);
Done    := (_exec = E_ExecState.DONE);
Error   := (_exec = E_ExecState.ERROR);
Aborted := (_exec = E_ExecState.ABORTED);
ErrorID := TO_DWORD(_diag.ReasonCode);

// §6.9(a)/§3.10(a') — refresh the data mirror: properties are invisible to the
// OPC UA namespace, so everything the HMI binds is published here as DATA
Status.ModuleType  := ModuleType;
Status.State       := _exec;
Status.FaultActive := (_exec = E_ExecState.ERROR);
Status.Diagnostic  := _diag;
_M_PublishStatus();              // tier-specific overlay after the common mirror is final

// A manual command is a one-shot use of the same PLCopen lifecycle. Keep the
// terminal state visible for this scan, then drop Execute for next-scan reset.
IF _manualActive AND ((_exec = E_ExecState.DONE) OR (_exec = E_ExecState.ERROR) OR (_exec = E_ExecState.ABORTED)) THEN
    Execute := FALSE;
    _manualActive := FALSE;
END_IF
Cyclic := TRUE;
END_METHOD

// Core §8.2/§6.9 — this node's first-out (composites override via rollup in the EM base)
METHOD GetFaultSummary : ST_Diagnostic
GetFaultSummary := _diag;
END_METHOD

// Core §3.14 hook — optional override: device-safe abort action.
// Override contract (Core §3.14.2): call SUPER^.OnAbort() FIRST and keep its return.
METHOD PROTECTED OnAbort : DINT
_exec := E_ExecState.ABORTED;
_step := 0;
OnAbort := 0;
END_METHOD

// Core §3.14 — optional error-state abort/recovery action. ERROR remains latched
// until Execute drops. Overrides call SUPER^.OnAbortInError() first.
METHOD PROTECTED OnAbortInError : DINT
OnAbortInError := 0;
END_METHOD

// Core §3.14 — first operational scan, after Setup/recipe load.
// Overrides call SUPER^.OnInit() first and propagate its return.
METHOD PROTECTED OnInit : DINT
OnInit := 0;
END_METHOD

// Core §3.14 hook — optional override: per-scan background management (idempotent,
// no direct outputs). Override contract: call SUPER^.OnCyclic() FIRST, keep return.
METHOD PROTECTED OnCyclic : DINT
OnCyclic := 0;
END_METHOD

// Core §3.14 hook — one-shot on each accepted Execute rising edge, after OnInit
// and before OnCyclic/_M_Dispatch. Overrides call SUPER^.OnCommandStart() first.
// Use for command-local wiring/reset only; process behavior belongs in dispatch.
METHOD PROTECTED OnCommandStart : DINT
OnCommandStart := 0;
END_METHOD

// Core §3.8 — types with ParCfg load into staging here.
METHOD PrepareRecipe : BOOL
VAR_INPUT
    Model : ST_ModelId;
END_VAR
PrepareRecipe := TRUE;
END_METHOD

METHOD CommitRecipe
END_METHOD

METHOD AbortRecipe
END_METHOD

// Core §3.2 — generic DINT command path; the catalog is the supported set.
// Concrete dispatch consumes the inherited manual request, so typed/generic/HMI
// paths share validation, timing, interlocks, and the PLCopen lifecycle.
METHOD ExecuteCommand : BOOL
VAR_INPUT
    Command : DINT;
END_VAR
ExecuteCommand := ManualCommand(Value := Command);
END_METHOD

// Core §3.2/§6.1 — method form of the inherited abort route.
METHOD AbortCommand : BOOL
AbortCommand := FALSE;
IF _exec <> E_ExecState.BUSY THEN
    RETURN;
END_IF
OnAbort();
_exec := E_ExecState.ABORTED;
_step := 0;
AbortCommand := TRUE;
END_METHOD

METHOD PROTECTED _M_ClearDiag
_diag.ReasonCode  := E_Reason.NONE;
_diag.Description := '';
_diag.IoTag := '';
_diag.IoAddress := '';
END_METHOD

// Core §6.1 — successful completion (the concrete type publishes OutCmd before calling)
METHOD PROTECTED _M_Complete
_exec := E_ExecState.DONE;
_step := 0;
_M_ClearDiag();
END_METHOD

// Core §2.2 — THE extension point: the type's CASE _step device logic,
// calling _M_Fault / _M_FaultDiag / _M_Complete.
METHOD PROTECTED ABSTRACT _M_Dispatch
END_METHOD

// Core §6.9 — stamp the first-out reason and hold in ERROR
METHOD PROTECTED _M_Fault
VAR_INPUT
    Reason : E_Reason;
    Text   : STRING(255);
END_VAR
_diag.ReasonCode  := Reason;
_diag.Description := Text;
_diag.SourcePath  := _name;
_diag.IoTag       := '';
_diag.IoAddress   := '';
_diag.Severity    := E_Severity.MED;
_diag.Category    := E_Category.PROCESS;
_diag.Since       := F_Now();       // synchronized clock (Core §2.7)
_exec := E_ExecState.ERROR;
_step := 0;
END_METHOD

// Core §8.2 — adopt a ready-made diagnostic verbatim (rollup / connector reason)
METHOD PROTECTED _M_FaultDiag
VAR_INPUT
    Diag : ST_Diagnostic;
END_VAR
_diag := Diag;
_exec := E_ExecState.ERROR;
_step := 0;
END_METHOD

// called from the concrete type's Setup (Core §3.11); Name = browse path (Core §4.8)
METHOD PROTECTED _M_SetName
VAR_INPUT
    Name : STRING(80);
END_VAR
_name := Name;
Status.Name := Name;   // mirror (§3.10(a'))
END_METHOD

// Core §8.11.4(a) — fold the finished command into its timing row (find-or-allocate)
METHOD PRIVATE _M_RecordCmdTiming
VAR_INPUT
    DurMs : DWORD;
END_VAR
VAR
    i, slot : INT;
END_VAR
Timing.LastCmdTime := DWORD_TO_TIME(DurMs);
slot := 0;
FOR i := 1 TO PL_Fraktal.MAX_CMD_STATS DO
    IF (Timing.Rows[i].Count > 0) AND (Timing.Rows[i].Id = _cmdId) THEN
        slot := i;
        EXIT;
    ELSIF (slot = 0) AND (Timing.Rows[i].Count = 0) THEN
        slot := i;
    END_IF
END_FOR
IF slot = 0 THEN
    Timing.Truncated := TRUE;        // fixed array, never grown at runtime (§8.11.4(e))
ELSE
    Timing.Rows[slot].Id    := _cmdId;
    Timing.Rows[slot].Label := _cmdLabel;
    F_TimingUpdate(Row := Timing.Rows[slot], DurMs := DurMs);
END_IF
END_METHOD

// Core §8.11.4(a) — the ONE line a type adds for a per-command breakdown:
//   _M_TagCommand(TO_DINT(Command), '<label>');   (idempotent; scaffold includes it)
METHOD PROTECTED _M_TagCommand
VAR_INPUT
    Id    : DINT;
    Label : STRING(120);
END_VAR
_cmdId    := Id;
    _cmdLabel := Label;
END_METHOD

// Optional localizable HMI metadata; keys only, never operator prose.
METHOD PROTECTED _M_SetPresentation
VAR_INPUT
    DisplayNameKey : STRING(160);
    DescriptionKey : STRING(160);
END_VAR
Status.DisplayNameKey := DisplayNameKey;
Status.DescriptionKey := DescriptionKey;
END_METHOD

// Core §8.8 band-extensibility: fault with a per-type band code (DINT constant).
// E_Reason is deliberately non-strict, so the numeric assignment is contract, not a cast trick.
METHOD PROTECTED _M_FaultN
VAR_INPUT
    Code : DINT;          // registered band code (Core §8.8 registry)
    Text : STRING(255);
END_VAR
_diag.ReasonCode  := Code;    // non-strict enum accepts the band value (Core §8.8)
_diag.Description := Text;
_diag.SourcePath  := _name;
_diag.IoTag       := '';
_diag.IoAddress   := '';
_diag.Severity    := E_Severity.MED;
_diag.Category    := E_Category.PROCESS;
_diag.Since       := F_Now();
_exec := E_ExecState.ERROR;
_step := 0;
END_METHOD

// Type-band fault with the implicated schematic tag and terminal location.
METHOD PROTECTED _M_FaultIoN
VAR_INPUT
    Code : DINT;
    Text : STRING(255);
    IoTag : STRING(80);
    IoAddress : STRING(80);
END_VAR
_M_FaultN(Code := Code, Text := Text);
_diag.IoTag := IoTag;
_diag.IoAddress := IoAddress;
END_METHOD

PROPERTY FaultActive : BOOL
GET
FaultActive := (_exec = E_ExecState.ERROR);
END_GET
END_PROPERTY

PROPERTY ModuleType : E_ModuleType
GET
ModuleType := E_ModuleType.NONE;
END_GET
END_PROPERTY

PROPERTY Name : STRING(80)
GET
Name := _name;
END_GET
END_PROPERTY

PROPERTY State : E_ExecState
GET
State := _exec;
END_GET
END_PROPERTY

// §7.6.1 — register one manual command in the catalog (call in the module's init).
// Idempotent by Value: re-publishing a Value updates its label.
METHOD PROTECTED _M_PublishCommand
VAR_INPUT
    Value : DINT;
    Label : STRING(120);
END_VAR
VAR
    i : INT;
END_VAR
FOR i := 1 TO CatalogCount DO
    IF Catalog[i].Value = Value THEN
        Catalog[i].Label := Label;
        RETURN;
    END_IF
END_FOR
IF CatalogCount >= PL_Fraktal.MAX_CMD_CATALOG THEN
    RETURN;
END_IF
CatalogCount := CatalogCount + 1;
Catalog[CatalogCount].Value := Value;
Catalog[CatalogCount].Label := Label;
END_METHOD

// §7.6.1 — apply a manual command, routed THROUGH the normal command surface so
// interlocks/first-out/timing still apply (§3.2). The owning Unit is the single
// gate: it calls this ONLY after verifying MANUAL mode (§3.4) + MANUAL access
// (§7.7) and logs the §8.3 event. §7.6 Release<Function> is enforced by the
// module's own _M_Dispatch. Concrete modules read _manualReq/_manualCmd there.
METHOD ManualCommand : BOOL
VAR_INPUT
    Value : DINT;
END_VAR
VAR
    i : INT;
    supported : BOOL;
END_VAR
ManualCommand := FALSE;
FOR i := 1 TO CatalogCount DO
    IF Catalog[i].Value = Value THEN
        supported := TRUE;
        EXIT;
    END_IF
END_FOR
IF NOT supported THEN
    RETURN;                              // reject values outside the published set (§5.6)
END_IF
IF (_exec <> E_ExecState.READY) OR Execute OR _manualActive THEN
    RETURN;
END_IF
_manualCmd := Value;
_manualReq := TRUE;                       // consumed by the module's _M_Dispatch
_manualActive := TRUE;
Execute := TRUE;                          // rising edge enters the inherited lifecycle
ManualCommand := TRUE;
END_METHOD

// Called after the common Status mirror refresh. Derived tiers may overlay data.
METHOD PROTECTED _M_PublishStatus
;
END_METHOD

// §3.10.1 — set the module's asset identity once, at Setup. Not HMI-writable;
// identity, not configuration (deliberately outside §3.8/§7.7).
METHOD SetNameplate : BOOL
VAR_INPUT
    Plate : ST_Nameplate;
END_VAR
Nameplate := Plate;
SetNameplate := TRUE;
END_METHOD

// §3.10.2 I_ConfigSource — export the base-owned static facets this module
// deliberately keeps off the cyclic OPC UA tree. Item fragments reproduce the
// server's array naming so the HMI rebuilds the exact browse paths generically.
// A type with additional static data overrides, calls SUPER^ first, appends.
METHOD M_AppendConfig : BOOL
VAR_INPUT
    Pager : REFERENCE TO FB_ConfigPager;
END_VAR
VAR
    i    : INT;
    item : STRING(255);
END_VAR
M_AppendConfig := TRUE;
Pager.M_AppendNumber(Scope := Status.Name, Item := 'CatalogCount',
    Number := TO_DINT(CatalogCount));
FOR i := 1 TO CatalogCount DO
    item := CONCAT('Catalog/Catalog[', CONCAT(TO_STRING(i), ']/Value'));
    Pager.M_AppendNumber(Scope := Status.Name, Item := item, Number := Catalog[i].Value);
    item := CONCAT('Catalog/Catalog[', CONCAT(TO_STRING(i), ']/Label'));
    Pager.M_Append(Scope := Status.Name, Item := item, ValueText := Catalog[i].Label);
END_FOR
END_METHOD

END_FUNCTION_BLOCK

// ---- BaseClasses/FB_CycleProfiler.TcPOU
// Core §8.11.4(b)/(f) — the cycle-time profile, fed by the step record the chain
// already keeps for §6.9: StepChanged() from _M_SetStep (with the step's time class,
// WORK by default), CycleComplete() at the finish step (§8.11.1 marker). Application
// steps add NOTHING except one enum on genuine wait steps. The step-chain / Unit
// base (M2) calls both automatically; until then a Unit wires the two calls once
// (Annex C §C.6). Fixed-size, no runtime allocation (Core §8.11.4(e)).
FUNCTION_BLOCK FB_CycleProfiler
VAR_OUTPUT
    Current        : ST_CycleProfile;   // cycle in progress (live waterfall)
    LastCycle      : ST_CycleProfile;   // last completed cycle — the HMI chart source
    StepStats      : ARRAY[1..PL_Fraktal.MAX_PROFILE_STEPS] OF ST_TimingRow;  // per-StepNo aggregates
    StatsTruncated : BOOL;
    // §8.11.1 throughput markers + §8.11.4 trend ring (the cycle-time ANALYSIS source:
    // per-cycle work/wait-class totals, charted by the HMI to explain increases)
    LastCycleTime  : TIME;
    MinCycleTime   : TIME;              // rolling minimum since reset (the demonstrated best)
    History        : ARRAY[1..PL_Fraktal.MAX_CYCLE_HISTORY] OF ST_CycleSummary;
    HistoryHead    : INT;               // newest entry (0 = none yet)
    // §8.11.4(d) — degradation is data: WorkTime drifting beyond Baseline*(1+BandPct)
    // pulses DegradedTrig for ONE call so the owner raises the maintenance event once.
    BaselineWorkMs : UDINT;             // 0 = degradation watch off (§3.8 config)
    DegradedBandPct: UDINT := 20;       // allowed drift above baseline, percent
    DegradedTrig   : BOOL;
    DegradedWorkMs : UDINT;             // the WorkTime that tripped the band (for the event text)
END_VAR
VAR
    _running      : BOOL;
    _openNo       : INT;
    _openName     : STRING(80);
    _openClass    : E_TimeClass;
    _openExpected : TIME;
    _openStartMs  : DWORD;
    _openStartDt  : DT;
    _cycleStartMs : DWORD;
    _degraded     : BOOL;               // latched: one event per excursion, not per cycle
END_VAR

// no cyclic body — event-driven via StepChanged/CycleComplete

// fold the open step into the profile, the class split, and the aggregates
METHOD PRIVATE _M_CloseOpen
VAR_INPUT
    NowMs : DWORD;
END_VAR
VAR
    dur  : DWORD;
    i    : INT;
    slot : INT;
END_VAR
IF _openNo = 0 THEN
    RETURN;
END_IF
dur := NowMs - _openStartMs;                                // wrap-safe (TC3 §8.11)

// (1) ordered waterfall entry
IF Current.NSteps < PL_Fraktal.MAX_PROFILE_STEPS THEN
    Current.NSteps := Current.NSteps + 1;
    Current.Steps[Current.NSteps].StepNo   := _openNo;
    Current.Steps[Current.NSteps].StepName := _openName;
    Current.Steps[Current.NSteps].TimeClass:= _openClass;
    Current.Steps[Current.NSteps].Started  := _openStartDt;
    Current.Steps[Current.NSteps].Duration := DWORD_TO_TIME(dur);
    Current.Steps[Current.NSteps].Expected := _openExpected;
ELSE
    Current.Truncated := TRUE;
END_IF

// (2) time-class split (§8.11.4(f)) — WorkTime/WaitTime derive from this at cycle close
Current.ByClass[TO_INT(_openClass)] := Current.ByClass[TO_INT(_openClass)] + DWORD_TO_TIME(dur);

// (3) per-StepNo aggregate (find-or-allocate; fixed array, Core §8.11.4(e))
slot := 0;
FOR i := 1 TO PL_Fraktal.MAX_PROFILE_STEPS DO
    IF (StepStats[i].Count > 0) AND (StepStats[i].Id = _openNo) THEN
        slot := i;
        EXIT;
    ELSIF (slot = 0) AND (StepStats[i].Count = 0) THEN
        slot := i;
    END_IF
END_FOR
IF slot = 0 THEN
    StatsTruncated := TRUE;
ELSE
    StepStats[slot].Id        := _openNo;
    StepStats[slot].Label     := _openName;
    StepStats[slot].TimeClass := _openClass;
    F_TimingUpdate(Row := StepStats[slot], DurMs := dur);
END_IF
END_METHOD

// §8.11.1 — discard the OPEN cycle without publishing it: a stop accepted at the
// between-cycles wait must not count a wait-only fragment as a production cycle
// (it would poison MinCycleTime and the trend). Aggregates keep completed cycles.
METHOD CycleAbandon : BOOL
_running := FALSE;
_openNo := 0;
CycleAbandon := TRUE;
END_METHOD

// close the open step and publish the cycle (call at the finish step, §8.11.1).
// Publishes WorkTime = ByClass[WORK] — the real cycle time (§8.11.4(f)).
METHOD CycleComplete : BOOL
VAR
    nowMs : DWORD;
END_VAR
IF NOT _running THEN
    CycleComplete := FALSE;
    RETURN;
END_IF
nowMs := TIME_TO_DWORD(TIME());
_M_CloseOpen(nowMs);
Current.Total    := DWORD_TO_TIME(nowMs - _cycleStartMs);   // wrap-safe (TC3 §8.11)
Current.WorkTime := Current.ByClass[TO_INT(E_TimeClass.WORK)];
Current.WaitTime := Current.Total - Current.WorkTime;
Current.CycleNo  := LastCycle.CycleNo + 1;
LastCycle := Current;

// §8.11.1 throughput markers
LastCycleTime := Current.Total;
IF (MinCycleTime = T#0S) OR (Current.Total < MinCycleTime) THEN
    MinCycleTime := Current.Total;
END_IF

// §8.11.4 trend ring — per-cycle class split for the HMI's cause analysis
HistoryHead := (HistoryHead MOD PL_Fraktal.MAX_CYCLE_HISTORY) + 1;
History[HistoryHead].CycleNo  := Current.CycleNo;
History[HistoryHead].Started  := Current.Started;
History[HistoryHead].Total    := Current.Total;
History[HistoryHead].WorkTime := Current.WorkTime;
History[HistoryHead].WaitTime := Current.WaitTime;
History[HistoryHead].ByClass  := Current.ByClass;

// §8.11.4(d) — degradation watch on WORK time (waits are attributed, not drift).
// One-call trigger, latched per excursion; recovery below the band rearms it.
DegradedTrig := FALSE;
DegradedWorkMs := TIME_TO_DWORD(Current.WorkTime);
IF BaselineWorkMs > 0 THEN
    IF DegradedWorkMs * 100 > BaselineWorkMs * (100 + DegradedBandPct) THEN
        IF NOT _degraded THEN
            _degraded := TRUE;
            DegradedTrig := TRUE;
        END_IF
    ELSE
        _degraded := FALSE;
    END_IF
END_IF

_running := FALSE;
_openNo  := 0;
CycleComplete := TRUE;
END_METHOD

// Configure the recipe-owned WORK-time reference through the profiler owner.
// BaselineWorkMs is published read-only; TwinCAT therefore rejects assignment
// through a parent FB's published Profiler output. Zero disables the watch.
METHOD M_SetBaselineWork : BOOL
VAR_INPUT
    WorkMs : UDINT;
END_VAR
BaselineWorkMs := WorkMs;
DegradedTrig := FALSE;
_degraded := FALSE;
M_SetBaselineWork := TRUE;
END_METHOD

// deliberate, LOGGED action only (Core §8.11.2) — the caller raises the event
METHOD ResetStats : BOOL
VAR
    i     : INT;
    empty : ST_TimingRow;
    emptySummary : ST_CycleSummary;
END_VAR
FOR i := 1 TO PL_Fraktal.MAX_PROFILE_STEPS DO
    StepStats[i] := empty;
END_FOR
FOR i := 1 TO PL_Fraktal.MAX_CYCLE_HISTORY DO
    History[i] := emptySummary;
END_FOR
HistoryHead := 0;
LastCycleTime := T#0S;
MinCycleTime := T#0S;
_degraded := FALSE;
StatsTruncated := FALSE;
LastCycle.CycleNo := 0;
ResetStats := TRUE;
END_METHOD

// call on every step change — _M_SetStep already has StepNo/StepName (§6.5).
// Class defaults to WORK; only genuine wait steps pass a wait class (§8.11.4(f)).
METHOD StepChanged : BOOL
VAR_INPUT
    StepNo   : INT;
    StepName : STRING(120);
    TimeClass    : E_TimeClass;
    Expected : TIME;                   // §8.11.4(c) — declared guard, drawn vs actual
END_VAR
VAR
    nowMs : DWORD;
    i     : INT;
END_VAR
IF _running AND (StepNo = _openNo) THEN
    _openClass := TimeClass;               // same step refreshed — class may be (re)declared
    _openExpected := Expected;
    StepChanged := TRUE;
    RETURN;
END_IF
nowMs := TIME_TO_DWORD(TIME());
IF NOT _running THEN
    _running := TRUE;                  // first step opens the cycle (§8.11.1 start marker)
    _cycleStartMs := nowMs;
    Current.Started   := F_Now();
    Current.NSteps    := 0;
    Current.Truncated := FALSE;
    FOR i := 0 TO 4 DO
        Current.ByClass[i] := T#0S;    // reset the class split for the new cycle
    END_FOR
ELSE
    _M_CloseOpen(nowMs);
END_IF
_openNo      := StepNo;
_openName    := StepName;
_openClass   := TimeClass;
_openExpected := Expected;
_openStartMs := nowMs;
_openStartDt := F_Now();
StepChanged := TRUE;
END_METHOD

END_FUNCTION_BLOCK

// ---- BaseClasses/FB_CompositeModuleBase.TcPOU
// Core §2.2 / §8.2 — CM lifecycle + child registry + first-out rollup.
// An EM type registers its children in Setup (_M_Register), ticks them every scan
// (_M_TickChildren, so status stays live whether or not a command runs — Annex B),
// and adopts the first faulted child's diagnostic verbatim (_M_RollupFault).
FUNCTION_BLOCK ABSTRACT FB_CompositeModuleBase EXTENDS FB_ModuleBase
VAR
    {attribute 'OPC.UA.DA' := '0'}
    _children : ARRAY[1..PL_Fraktal.MAX_EM_CHILDREN] OF I_Module;
    _nChild   : INT;
END_VAR

Cyclic();

// called from the type's Setup (Core §3.11); bounds-checked per Core §5.6
METHOD PROTECTED _M_Register : BOOL
VAR_INPUT
    Child : I_Module;
END_VAR
IF (Child = 0) OR (_nChild >= PL_Fraktal.MAX_EM_CHILDREN) THEN
    _M_Register := FALSE;
    RETURN;
END_IF
_nChild := _nChild + 1;
_children[_nChild] := Child;
_M_Register := TRUE;
END_METHOD

METHOD PrepareRecipe : BOOL
VAR_INPUT
    Model : ST_ModelId;
END_VAR
VAR
    i, j : INT;
END_VAR
PrepareRecipe := TRUE;
FOR i := 1 TO _nChild DO
    IF (_children[i] <> 0) AND_THEN NOT _children[i].PrepareRecipe(Model := Model) THEN
        PrepareRecipe := FALSE;
        FOR j := 1 TO i DO
            IF _children[j] <> 0 THEN _children[j].AbortRecipe(); END_IF
        END_FOR
        RETURN;
    END_IF
END_FOR
END_METHOD

METHOD CommitRecipe
VAR
    i : INT;
END_VAR
FOR i := 1 TO _nChild DO
    IF _children[i] <> 0 THEN _children[i].CommitRecipe(); END_IF
END_FOR
END_METHOD

METHOD AbortRecipe
VAR
    i : INT;
END_VAR
FOR i := 1 TO _nChild DO
    IF _children[i] <> 0 THEN _children[i].AbortRecipe(); END_IF
END_FOR
END_METHOD

// Core §8.2 — adopt the FIRST faulted child's first-out (reason + child SourcePath)
METHOD PROTECTED _M_RollupFault : BOOL
VAR
    i : INT;
END_VAR
_M_RollupFault := FALSE;
FOR i := 1 TO _nChild DO
    IF _children[i] <> 0 AND_THEN _children[i].FaultActive THEN
        _M_FaultDiag(_children[i].GetFaultSummary());
        _M_RollupFault := TRUE;
        RETURN;
    END_IF
END_FOR
END_METHOD

// children always tick so their status stays live (Annex B §B.3)
METHOD PROTECTED _M_TickChildren
VAR
    i : INT;
END_VAR
FOR i := 1 TO _nChild DO
    IF _children[i] <> 0 THEN
        _children[i].Cyclic();
    END_IF
END_FOR
END_METHOD

PROPERTY ModuleType : E_ModuleType
GET
ModuleType := E_ModuleType.NONE;
END_GET
END_PROPERTY

// §3.10.2 — own facets first, then every registered child, depth-first in
// registration order so the manifest walk is deterministic across requests.
METHOD M_AppendConfig : BOOL
VAR_INPUT
    Pager : REFERENCE TO FB_ConfigPager;
END_VAR
VAR
    i    : INT;
    iCfg : I_ConfigSource;
END_VAR
M_AppendConfig := SUPER^.M_AppendConfig(Pager := Pager);
FOR i := 1 TO _nChild DO
    IF _children[i] <> 0 THEN
        IF __QUERYINTERFACE(_children[i], iCfg) THEN
            iCfg.M_AppendConfig(Pager := Pager);
        END_IF
    END_IF
END_FOR
END_METHOD

END_FUNCTION_BLOCK

// ---- BaseClasses/FB_UnitBase.TcPOU
// Core §2.2 lifecycle family, top tier: modes + cascade (§3.4/§3.7), Start/Stop
// mapped onto the §6.1 run command (§6 intro), the step chain (_M_SetStep/_M_Await,
// §6.5/§6.9(b)), the stall walk as a PENDING reason with instant rollup on an
// awaited module's Error (§6.9/§8.2), the §8.11.4 profiler wired in, and
// Starved/Blocked derived from the step's time class (§8.11.4(f)/§8.11.3).
// A Unit type overrides _M_Dispatch (its mode chain) + _M_Supports (+ §3.14 hooks).
FUNCTION_BLOCK ABSTRACT FB_UnitBase EXTENDS FB_CompositeModuleBase IMPLEMENTS I_Unit, I_SequenceHost
VAR_INPUT
    DecisionAnswer : INT;              // §6.11: chosen option index (0 = none yet)
    ReqControlOn   : BOOL;             // §9.8 HMI/data request; edge-consumed and access-gated
    ReqControlOff  : BOOL;
    HmiRequest     : ST_HmiRequest;     // §3.10/§14: arguments first, Sequence last
    {attribute 'OPC.UA.DA' := '0'}
    ControlDomain  : ST_ControlDomainStatus; // §9.8: optional shared cell/cage arrangement
END_VAR
VAR_OUTPUT
    Starved : BOOL;                    // §8.11.3 — derived from CurrentStep.Class
    Blocked : BOOL;
    Domain  : ST_ControlDomainStatus;  // §9.8 read-only publication of the assigned domain
    ControlOnRequest  : BOOL;          // one-scan request to the owning domain coordinator
    ControlOffRequest : BOOL;
END_VAR
VAR_OUTPUT
    Profiler    : FB_CycleProfiler;    // §8.11.4 — HMI chart source
    CurrentStep : ST_StepRecord;       // §6.5 — feeds §6.9 walk AND the profiler
    Pending     : ST_Diagnostic;       // live stall reason (Low) — NOT a fault (§6.9)
    Decision    : ST_DecisionRequest;  // §6.11 active request ('' Prompt = none)
    {attribute 'OPC.UA.DA' := '0'}
    StallTime   : TIME := T#30S;       // guard when the step declares no ExpectedTime
    Model       : ST_ModelId;          // §3.1b active model identity (published for HMI/MES/trace)
    // §3.10.2 — static catalogs served via the QUERY_CONFIG manifest, not cyclically
    {attribute 'OPC.UA.DA' := '0'}
    AvailableModelCount : INT;         // §3.8 optional discoverable model/recipe catalog
    {attribute 'OPC.UA.DA' := '0'}
    AvailableModels : ARRAY[1..PL_Fraktal.MAX_RECIPES] OF ST_ModelId;
    Part        : ST_PartContext;      // §3.16.1 live part context (Present=FALSE, Uid='' = none)
    AlarmLog    : FB_AlarmLog;         // §8.3 — active list + closed ring + Blocking
    Access      : FB_AccessManager;    // §7.7 — per-root session/policy (default: fully open)
    GoodCount   : UDINT;               // §8.11.2 — cycle verdict counters
    NokCount    : UDINT;
    ReworkCount : UDINT;
    NokReason   : E_Reason;            // §8.11.2 — last NOK's first-out attribution
    MachineState : E_MachineState;     // §8.11.3 — classified every scan (OEE/PackML/host)
    History     : ARRAY[1..PL_Fraktal.MAX_DIAG_RING] OF ST_Diagnostic;  // §6.9(a) ring (newest at HistoryHead)
    HistoryHead : INT;
    {attribute 'OPC.UA.DA' := '0'}
    ModePolicy  : ARRAY[0..PL_Fraktal.MODE_COUNT-1] OF ST_ModePolicy;    // §3.4.1 per-mode switch policy (station cfg; manifest-served)
    RunStyle    : E_RunStyle;          // §3.4.2 active run style (HMI-selectable; CONTINUOUS default)
    Oee         : ST_Oee;              // §8.5.1 accumulators + snapshot (published)
    OeeTrend    : ARRAY[1..PL_Fraktal.MAX_OEE_SAMPLES] OF ST_OeeSample; // §8.5.1 ring
    OeeTrendHead: INT;                 // newest sample index (0 = none yet)
    HmiResponse : ST_HmiResponse;
    ConfigRev   : UDINT;                // §3.10.2 manifest revision — HMI refetches on change
    ModeActivePublished : E_Mode;       // properties are not OPC UA-visible
    RunningPublished : BOOL;
    StopPendingPublished : BOOL;
    SupportedModesPublished : ARRAY[0..PL_Fraktal.MODE_COUNT-1] OF BOOL;
    SupportedRunStylesPublished : ARRAY[0..2] OF BOOL;
END_VAR
VAR
    _fTrig    : R_TRIG;
    _mode     : E_Mode;
    _modeReq  : E_Mode;
    _modePend : BOOL;
    _modeExitFirst : BOOL;
    _stopReq  : BOOL;
    {attribute 'OPC.UA.DA' := '0'}
    _awaits   : I_Module;              // module the current step awaits (0 = none)
    _faultEvt : INT;                   // open ERROR event slot in AlarmLog (0 = none)
    _tStall   : TON;
    _stepReq  : BOOL;                  // §3.4.2 pending single-step request (edge-consumed)
    _holdRun  : BOOL;                  // §3.4.2 HOLD_TO_RUN input held (NON-SAFETY, §9)
    _stepArm  : R_TRIG;
    _oeeLast  : TIME;                  // §8.5.1 last accumulation stamp
    _oeeSampMs: UDINT;                 // ms since last trend sample
    _hmiLastSequence : UDINT;
    {attribute 'OPC.UA.DA' := '0'}
    _configPager : FB_ConfigPager;     // §3.10.2 QUERY_CONFIG window writer
    {attribute 'OPC.UA.DA' := '0'}
    _carrier  : I_PartCarrier;         // §3.16.2 injected part carrier (0 = traceability off)
END_VAR

Cyclic();

// Core §7.8 helper — append one non-interlock reason (bounds-checked).
METHOD PROTECTED _M_AddReason
VAR_IN_OUT
    Report : ST_ReleaseReport;
END_VAR
VAR_INPUT
    Text : STRING(255);
    Reason : E_Reason;
    Kind : E_ReleaseKind;
END_VAR
IF Report.Count >= PL_Fraktal.MAX_RELEASE_REASONS THEN
    RETURN;
END_IF
Report.Count := Report.Count + 1;
Report.Reasons[Report.Count].Description := Text;
Report.Reasons[Report.Count].ReasonCode  := Reason;
Report.Reasons[Report.Count].SourcePath  := _name;
Report.Reasons[Report.Count].Kind        := Kind;
Report.Reasons[Report.Count].Bypassable  := FALSE;
END_METHOD

// Core §7.8 — concrete Units override to append the active mode's immediate
// entry/frontier records via PermIntlk.AppendFailed(SourcePath, Report). Future step waits
// stay in CurrentStep/Pending and are not blanket Start conditions. Base: nothing.
METHOD PROTECTED _M_AppendInterlocks
VAR_IN_OUT
    Report : ST_ReleaseReport;
END_VAR
;
END_METHOD

// Core §7.8 — target-aware hook for the MANUAL release rollup: a concrete Unit
// overrides to append the §7.6 Release<Function> conditions of the SPECIFIC target
// module. Base delegates to the Unit-level hook (non-breaking default).
METHOD PROTECTED _M_AppendManualInterlocks
VAR_INPUT
    TargetPath : STRING(255);
    Value : DINT;
END_VAR
VAR_IN_OUT
    Report : ST_ReleaseReport;
END_VAR
_M_AppendInterlocks(Report := Report);
END_METHOD

// §6.11 — publish a typed decision request (single active slot)
METHOD PROTECTED _M_AskDecision
VAR_INPUT
    Req : ST_DecisionRequest;
END_VAR
Decision := Req;
Decision.SourcePath := _name;
END_METHOD

// §6.9(b) — named plain-condition wait; returns the condition so steps read naturally
METHOD PROTECTED _M_Await : BOOL
VAR_INPUT
    Idx   : INT;
    Label : STRING(120);
    Ok    : BOOL;
END_VAR
IF (Idx >= 1) AND (Idx <= PL_Fraktal.MAX_STEP_CONDS) THEN
    CurrentStep.Conds[Idx].Label := Label;
    CurrentStep.Conds[Idx].Ok    := Ok;
END_IF
_M_Await := Ok;
END_METHOD

// §3.7 — offer the mode to child Units; a child may reject (graceful)
METHOD PROTECTED _M_CascadeMode
VAR_INPUT
    Mode : E_Mode;
END_VAR
VAR
    i  : INT;
    iu : I_Unit;
END_VAR
FOR i := 1 TO _nChild DO
    IF _children[i] <> 0 THEN
        IF __QUERYINTERFACE(_children[i], iu) THEN   // [TC3] capability query — TC3 §3.2
            iu.SetMode(Mode);
        END_IF
    END_IF
END_FOR
END_METHOD

METHOD PROTECTED _M_ClearPending
Pending.ReasonCode  := E_Reason.NONE;
Pending.Description := '';
END_METHOD

// call at the finish step (§8.11.1): publishes the profile; FALSE = stop granted
METHOD PROTECTED _M_EndOfCycle : BOOL
Profiler.CycleComplete();
IF _stopReq THEN
    _stopReq := FALSE;
    Execute := FALSE;
    _M_Complete();
    _M_EndOfCycle := FALSE;
ELSE
    _M_EndOfCycle := TRUE;
END_IF
END_METHOD

// §3.10/§14 — consume one committed OPC UA request exactly once.
METHOD PROTECTED _M_HandleHmiRequest
VAR
    modelId  : ST_ModelId;
    modeReq  : E_Mode;
    styleReq : E_RunStyle;
    gateReq  : E_GatedAction;
END_VAR
IF HmiRequest.Sequence = _hmiLastSequence THEN
    RETURN;
ELSE
    _hmiLastSequence := HmiRequest.Sequence;
END_IF

HmiResponse.Accepted := FALSE;
HmiResponse.Diagnostic := '';
HmiResponse.Report.Count := 0;
HmiResponse.Report.Released := FALSE;

CASE HmiRequest.Kind OF
    E_HmiRequestKind.LOGIN:
        HmiResponse.Accepted := Access.RequestLogin(User := HmiRequest.User, Secret := HmiRequest.Secret);
    E_HmiRequestKind.LOGOUT:
        HmiResponse.Accepted := Access.RequestLogout();
    E_HmiRequestKind.SET_MODE:
        IF (HmiRequest.IntValue >= 0) AND (HmiRequest.IntValue < PL_Fraktal.MODE_COUNT) THEN
            modeReq := HmiRequest.IntValue;
            HmiResponse.Accepted := SetMode(Mode := modeReq);
        ELSE
            HmiResponse.Diagnostic := 'std.error.unsupportedModeRequest';
        END_IF
    E_HmiRequestKind.SET_MODEL:
        modelId.ModelCode := HmiRequest.TextValue;
        HmiResponse.Accepted := SetModel(Id := modelId);
    E_HmiRequestKind.START:
        HmiResponse.Accepted := Start();
    E_HmiRequestKind.STOP:
        HmiResponse.Accepted := Stop();
    E_HmiRequestKind.CONTROL_ON:
        ReqControlOn := TRUE;
        ReqControlOff := FALSE;
        HmiResponse.Accepted := TRUE;
    E_HmiRequestKind.CONTROL_OFF:
        ReqControlOff := TRUE;
        ReqControlOn := FALSE;
        HmiResponse.Accepted := TRUE;
    E_HmiRequestKind.OPERATOR_RESET:
        HmiResponse.Accepted := OperatorReset();
    E_HmiRequestKind.DECISION_ANSWER:
        DecisionAnswer := TO_INT(HmiRequest.IntValue);
        HmiResponse.Accepted := TRUE;
    E_HmiRequestKind.MANUAL_COMMAND:
        HmiResponse.Accepted := ManualCommandTo(TargetPath := HmiRequest.TargetPath, Value := HmiRequest.IntValue);
    E_HmiRequestKind.SET_RUN_STYLE:
        IF (HmiRequest.IntValue >= 0) AND (HmiRequest.IntValue <= 2) THEN
            styleReq := HmiRequest.IntValue;
            HmiResponse.Accepted := SetRunStyle(Style := styleReq);
        ELSE
            HmiResponse.Diagnostic := 'std.error.unsupportedRunStyleRequest';
        END_IF
    E_HmiRequestKind.STEP_REQUEST:
        HmiResponse.Accepted := StepRequest();
    E_HmiRequestKind.SET_HOLD_RUN:
        HmiResponse.Accepted := SetHoldRun(Held := HmiRequest.BoolValue);
    E_HmiRequestKind.RELEASE_START:
        ReleaseReportStart(Report := HmiResponse.Report);
        HmiResponse.Accepted := TRUE;
    E_HmiRequestKind.RELEASE_MANUAL:
        ReleaseReportManual(TargetPath := HmiRequest.TargetPath, Value := HmiRequest.IntValue,
            Report := HmiResponse.Report);
        HmiResponse.Accepted := TRUE;
    E_HmiRequestKind.RELEASE_ACTION:
        IF (HmiRequest.IntValue >= 0) AND (HmiRequest.IntValue <= 10) THEN
            gateReq := HmiRequest.IntValue;
            ReleaseReportAction(Gate := gateReq, Report := HmiResponse.Report);
            HmiResponse.Accepted := TRUE;
        ELSE
            HmiResponse.Diagnostic := 'std.error.unsupportedGatedActionRequest';
        END_IF
    E_HmiRequestKind.RESET_OEE:
        HmiResponse.Accepted := ResetOee();
    E_HmiRequestKind.WRITE_CONFIG:
        HmiResponse.Accepted := _M_RouteConfigWrite(TargetPath := HmiRequest.TargetPath,
            FieldName := HmiRequest.NameValue, TextValue := HmiRequest.TextValue);
        IF HmiResponse.Accepted THEN
            ConfigRev := ConfigRev + 1;    // §3.10.2 — manifest changed
        END_IF
    E_HmiRequestKind.SHELVE_ALARM:
        HmiResponse.Diagnostic := 'std.error.identityAlarmRequestNotSupported';
    E_HmiRequestKind.UNSHELVE_ALARM:
        HmiResponse.Diagnostic := 'std.error.identityAlarmRequestNotSupported';
    E_HmiRequestKind.FORCE_CHANNEL:
        HmiResponse.Accepted := _M_RouteForceChannel(ChannelPath := HmiRequest.TargetPath,
            Force := HmiRequest.BoolValue, BoolText := HmiRequest.TextValue,
            AnalogText := HmiRequest.NameValue);
    E_HmiRequestKind.QUERY_CONFIG:
        // §3.10.2 — serve one manifest page: re-walk the deterministic export
        // enumeration, storing only the requested window (no full buffer).
        IF _configPager.M_Setup(Target := ADR(HmiResponse.ConfigPage),
            PageIndex := TO_INT(HmiRequest.IntValue), Revision := ConfigRev) THEN
            M_AppendConfig(Pager := _configPager);
            _configPager.M_Finish();
            HmiResponse.Accepted := TRUE;
        ELSE
            HmiResponse.Diagnostic := 'std.error.hmiRequestRejected';
        END_IF
    E_HmiRequestKind.NONE:
        HmiResponse.Diagnostic := 'std.error.emptyHmiRequest';
ELSE
    HmiResponse.Diagnostic := 'std.error.unsupportedHmiRequest';
END_CASE

IF NOT HmiResponse.Accepted AND (HmiResponse.Diagnostic = '') THEN
    HmiResponse.Diagnostic := 'std.error.hmiRequestRejected';
ELSE
    HmiResponse.Diagnostic := HmiResponse.Diagnostic;
END_IF
HmiRequest.Secret := '';
HmiResponse.AckSequence := _hmiLastSequence;
END_METHOD

// §3.4.1/§3.14.4 — default per-mode switch policy. Station config (§3.8a) may
// overwrite ModePolicy[] after this. By FRAMEWORK DEFAULT a mode change while a
// sequence runs performs an IMMEDIATE software abort (E-stop-like, not a safety
// function, §3.14.4) — so Style defaults to IMMEDIATE. GRACEFUL completion is an
// opt-in: a Unit overrides OnModeExit to stop-after-cycle, or station config sets
// Style := GRACEFUL for a mode. Shield only governs acceptance while running.
METHOD PROTECTED _M_InitModePolicy
VAR
    i : INT;
END_VAR
FOR i := 0 TO PL_Fraktal.MODE_COUNT-1 DO
    ModePolicy[i].Shield := E_ModeSwitchShield.CONFIRM;
    ModePolicy[i].Style  := E_ModeSwitchStyle.IMMEDIATE;
END_FOR
// Setup modes a running machine may not leave without an explicit Stop first.
ModePolicy[TO_INT(E_Mode.CHANGEOVER)].Shield := E_ModeSwitchShield.BLOCKED_WHILE_RUNNING;
ModePolicy[TO_INT(E_Mode.CALIBRATION)].Shield:= E_ModeSwitchShield.BLOCKED_WHILE_RUNNING;
// HOME and MANUAL are freely interruptible; both inherit the IMMEDIATE default.
ModePolicy[TO_INT(E_Mode.HOME)].Shield       := E_ModeSwitchShield.INTERRUPTIBLE;
ModePolicy[TO_INT(E_Mode.MANUAL)].Shield     := E_ModeSwitchShield.INTERRUPTIBLE;
END_METHOD

// §8.5.1 — pure recompute of A/P/Q/OEE from the accumulators (testable in isolation).
// Invalid factors are OMITTED from the product, never assumed 100% (O7).
METHOD PROTECTED _M_OeeCompute
VAR
    total : UDINT;
    denomA: UDINT;
END_VAR
denomA := Oee.RunMs + Oee.DownMs;
Oee.AvailValid := denomA > 0;
IF Oee.AvailValid THEN
    Oee.Availability := UDINT_TO_REAL(Oee.RunMs) / UDINT_TO_REAL(denomA);
ELSE
    Oee.Availability := 0.0;
END_IF
Oee.PerfValid := (Oee.IdealCycleMs > 0) AND (Oee.RunMs > 0);
IF Oee.PerfValid THEN
    Oee.Performance := UDINT_TO_REAL(Oee.IdealCycleMs) * UDINT_TO_REAL(GoodCount + NokCount)
                       / UDINT_TO_REAL(Oee.RunMs);
    IF Oee.Performance > 1.0 THEN
        Oee.Performance := 1.0;          // faster than ideal caps at 100% (standard practice)
    END_IF
ELSE
    Oee.Performance := 0.0;
END_IF
total := GoodCount + NokCount;
Oee.QualValid := total > 0;
IF Oee.QualValid THEN
    Oee.Quality := UDINT_TO_REAL(GoodCount) / UDINT_TO_REAL(total);
ELSE
    Oee.Quality := 0.0;
END_IF
// product of VALID factors only; OEE valid iff at least one factor is valid
Oee.Oee := 1.0;
Oee.OeeValid := FALSE;
IF Oee.AvailValid THEN Oee.Oee := Oee.Oee * Oee.Availability; Oee.OeeValid := TRUE; END_IF
IF Oee.PerfValid  THEN Oee.Oee := Oee.Oee * Oee.Performance;  Oee.OeeValid := TRUE; END_IF
IF Oee.QualValid  THEN Oee.Oee := Oee.Oee * Oee.Quality;      Oee.OeeValid := TRUE; END_IF
IF NOT Oee.OeeValid THEN
    Oee.Oee := 0.0;
END_IF
END_METHOD

// §8.5.1 — attribute elapsed time to run/down/idle, recompute factors, sample ring.
METHOD PROTECTED _M_OeeUpdate
VAR
    currentTime : TIME;
    deltaMs     : UDINT;
END_VAR
currentTime := TIME();                 // monotonic duration clock
IF _oeeLast = T#0S THEN
    _oeeLast := currentTime;
    RETURN;
END_IF
deltaMs := TIME_TO_UDINT(currentTime) - TIME_TO_UDINT(_oeeLast); // wrap-safe on UDINT subtraction
_oeeLast := currentTime;
IF _exec = E_ExecState.BUSY THEN
    Oee.RunMs := Oee.RunMs + deltaMs;
ELSIF (_exec = E_ExecState.ERROR) OR AlarmLog.Blocking THEN
    Oee.DownMs := Oee.DownMs + deltaMs;
ELSE
    Oee.IdleMs := Oee.IdleMs + deltaMs;
END_IF
_M_OeeCompute();
_oeeSampMs := _oeeSampMs + deltaMs;
IF _oeeSampMs >= PL_Fraktal.OEE_SAMPLE_MS THEN
    _oeeSampMs := 0;
    OeeTrendHead := (OeeTrendHead MOD PL_Fraktal.MAX_OEE_SAMPLES) + 1;
    OeeTrend[OeeTrendHead].Availability := Oee.Availability;
    OeeTrend[OeeTrendHead].Performance  := Oee.Performance;
    OeeTrend[OeeTrendHead].Quality      := Oee.Quality;
    OeeTrend[OeeTrendHead].Oee          := Oee.Oee;
    OeeTrend[OeeTrendHead].OeeValid     := Oee.OeeValid;
END_IF
END_METHOD

// §3.16.3 EVENT_PART_PROCESSING_ABORTED — the part leaves without a valid result
// (fault, abort, manual removal). Called automatically on Unit ERROR entry.
METHOD PROTECTED _M_PartAborted
IF (_carrier = 0) OR NOT Part.Present THEN
    RETURN;
END_IF
Part.Result.Verdict := E_Verdict.NONE;
_M_PartEvent(Reason := E_Reason.EVENT_PART_PROCESSING_ABORTED,
    Text := 'std.event.partAborted: ');
Part.Present := FALSE;
END_METHOD

// §3.16.3 — one canonical part-lifecycle event: instant come+gone MESSAGE ring entry.
METHOD PRIVATE _M_PartEvent
VAR_INPUT
    Reason : E_Reason;
    Text : STRING(255);
END_VAR
VAR
    slot : INT;
    txt : STRING(255);
END_VAR
txt := CONCAT(Text, Part.Uid);
slot := AlarmLog.Raise(Reason := Reason, Text := txt, Source := _name,
    Severity := E_Severity.LOW, Category := E_Category.PROCESS,
    ResetClass := E_ResetClass.AUTO_RESET);
IF slot > 0 THEN
    AlarmLog.Gone(Slot := slot);
END_IF
END_METHOD

// §3.16.3 EVENT_PART_PROCESSED — stamp the verdict, write the carrier FIRST
// (result-before-event contract), then raise the event. The Uid and result stay
// published until the next part so the HMI shows the last outcome.
METHOD PROTECTED _M_PartProcessed : BOOL
VAR_INPUT
    Verdict : E_Verdict;
    Reason : E_Reason;
END_VAR
_M_PartProcessed := FALSE;
IF (_carrier = 0) OR NOT Part.Present THEN
    RETURN;
END_IF
Part.Result.Verdict := Verdict;
Part.Result.ReasonCode := Reason;
Part.Result.StationPath := _name;
Part.Result.Stamp := F_Now();
IF NOT _carrier.WriteResult(Ctx := Part) THEN
    _M_Fault(E_Reason.CARRIER_WRITE_FAILED, 'std.error.partCarrierWriteFailed');
    RETURN;
END_IF
// §8.11.2 — counters increment HERE, from the verdict; an NOK carries its
// first-out ReasonCode so scrap is analysable by cause (§8.8 vocabulary).
CASE Verdict OF
    E_Verdict.OK:     CountGood();
    E_Verdict.NOK:    CountNok();    NokReason := Reason;
    E_Verdict.REWORK: CountRework();
ELSE
    ;                                // NONE: no count — the part left unjudged
END_CASE
_M_PartEvent(Reason := E_Reason.EVENT_PART_PROCESSED, Text := 'std.event.partProcessed: ');
Part.Present := FALSE;
_M_PartProcessed := TRUE;
END_METHOD

// §3.16.3 EVENT_PART_RECEIVED — confirm identity at station entry via the carrier.
// FALSE with a CARRIER_READ_FAILED fault on a failed read (never silent), FALSE
// silently when no carrier is configured (§3.9 feature selectability).
METHOD PROTECTED _M_PartReceived : BOOL
VAR
    i : INT;
END_VAR
_M_PartReceived := FALSE;
IF _carrier = 0 THEN
    RETURN;
END_IF
Part.Uid := '';                              // station entry = fresh identity read
IF NOT _carrier.ReadContext(Ctx := Part) THEN
    _M_Fault(E_Reason.CARRIER_READ_FAILED, 'std.error.partCarrierReadFailed');
    RETURN;
END_IF
Part.Result.Verdict := E_Verdict.NONE;       // this station's outcome starts empty
Part.Result.ReasonCode := E_Reason.NONE;
Part.Result.StationPath := _name;
FOR i := 1 TO PL_Fraktal.MAX_RESULTS DO
    Part.Result.Records[i].Name := '';
END_FOR
_M_PartEvent(Reason := E_Reason.EVENT_PART_RECEIVED, Text := 'std.event.partReceived: ');
_M_PartReceived := TRUE;
END_METHOD

// §3.16.1 — append one measured value to this part's result (test cells).
// FALSE when the bounded record table is full (RESULT_RECORD_REJECTED semantics).
METHOD PROTECTED _M_PartRecord : BOOL
VAR_INPUT
    RecordName : STRING(64);
    Value : LREAL;
    Minimum : LREAL;
    Maximum : LREAL;
    Target : LREAL;
    EngUnit : STRING(16);
END_VAR
VAR
    i : INT;
END_VAR
_M_PartRecord := FALSE;
IF NOT Part.Present THEN
    RETURN;
END_IF
FOR i := 1 TO PL_Fraktal.MAX_RESULTS DO
    IF Part.Result.Records[i].Name = '' THEN
        Part.Result.Records[i].Name := RecordName;
        Part.Result.Records[i].Value := Value;
        Part.Result.Records[i].Minimum := Minimum;
        Part.Result.Records[i].Maximum := Maximum;
        Part.Result.Records[i].Target := Target;
        Part.Result.Records[i].Unit := EngUnit;
        Part.Result.Records[i].InTol := (Maximum <= Minimum)
            OR ((Value >= Minimum) AND (Value <= Maximum));
        _M_PartRecord := TRUE;
        RETURN;
    END_IF
END_FOR
END_METHOD

// §3.16.3 EVENT_PART_PROCESSING_STARTED — the value-adding sequence begins.
METHOD PROTECTED _M_PartStarted
IF (_carrier = 0) OR NOT Part.Present THEN
    RETURN;
END_IF
_M_PartEvent(Reason := E_Reason.EVENT_PART_PROCESSING_STARTED,
    Text := 'std.event.partProcessingStarted: ');
END_METHOD

// §6.9/§3.10(a') — overlay the pending stall after the common mirror refresh.
METHOD PROTECTED _M_PublishStatus
SUPER^._M_PublishStatus();
// §8.11.4(f)/§8.11.3 — one declaration, two views. Derived AFTER dispatch so the
// wait class reflects the step record this scan just set, not the previous one.
Starved := (_exec = E_ExecState.BUSY) AND (CurrentStep.TimeClass = E_TimeClass.WAIT_UPSTREAM);
Blocked := (_exec = E_ExecState.BUSY) AND (CurrentStep.TimeClass = E_TimeClass.WAIT_DOWNSTREAM);
// §8.11.3 — classify into the fixed machine-state set (priority: fault first,
// then planned states, then line attribution, then producing/idle).
IF (_exec = E_ExecState.ERROR) OR AlarmLog.Blocking THEN
    MachineState := E_MachineState.DOWN;
ELSIF _mode = E_Mode.CHANGEOVER THEN
    MachineState := E_MachineState.CHANGEOVER;
ELSIF Blocked THEN
    MachineState := E_MachineState.BLOCKED;
ELSIF Starved THEN
    MachineState := E_MachineState.STARVED;
ELSIF _exec = E_ExecState.BUSY THEN
    MachineState := E_MachineState.PRODUCING;
ELSIF _stopReq OR (_exec = E_ExecState.ABORTED) THEN
    MachineState := E_MachineState.STOPPED;
ELSE
    MachineState := E_MachineState.IDLE;
END_IF
Status.ControlDomainId := ControlDomain.Id;
Domain := ControlDomain;
Safety := ControlDomain.Safety;             // read-only HMI mirror; ownership stays in domain
ControlPower := ControlDomain.ControlPower;
IF (_exec <> E_ExecState.ERROR) AND (Pending.ReasonCode <> E_Reason.NONE) THEN
    Status.Diagnostic := Pending;
END_IF
END_METHOD

// §6.9(a) — fixed ring, newest at HistoryHead; never allocates
METHOD PROTECTED _M_PushHistory
VAR_INPUT
    D : ST_Diagnostic;
END_VAR
HistoryHead := (HistoryHead MOD PL_Fraktal.MAX_DIAG_RING) + 1;
History[HistoryHead] := D;
END_METHOD

// §8.11.4(d)/§8.12 — a Low-severity maintenance event: informs planning, does not
// stop the cycle. Instant come+gone ring entry (the trend data lives in Profiler).
METHOD PROTECTED _M_RaiseMaintenance
VAR_INPUT
    Reason : E_Reason;
    Text : STRING(255);
END_VAR
VAR
    slot : INT;
END_VAR
slot := AlarmLog.Raise(Reason := Reason, Text := Text, Source := _name,
    Severity := E_Severity.LOW, Category := E_Category.SYSTEM,
    ResetClass := E_ResetClass.AUTO_RESET);
IF slot > 0 THEN
    AlarmLog.Gone(Slot := slot);
END_IF
END_METHOD

// Project/type override for published editable fields. Base fails closed.
METHOD PROTECTED _M_RouteConfigWrite : BOOL
VAR_INPUT
    TargetPath : STRING(255);
    FieldName  : STRING(160);
    TextValue  : STRING(255);
END_VAR
_M_RouteConfigWrite := FALSE;
END_METHOD

// Application override routes only approved outputs through its force gate.
METHOD PROTECTED _M_RouteForceChannel : BOOL
VAR_INPUT
    ChannelPath : STRING(255);
    Force       : BOOL;
    BoolText    : STRING(255);
    AnalogText  : STRING(160);
END_VAR
_M_RouteForceChannel := FALSE;
END_METHOD

// §7.6.1 — concrete Units override to map a target path to a child module and call
// its ManualCommand. Base returns FALSE (no commandable children).
METHOD PROTECTED _M_RouteManual : BOOL
VAR_INPUT
    TargetPath : STRING(255);
    Value : DINT;
END_VAR
_M_RouteManual := FALSE;
END_METHOD

// §6.5 — the ONE line per step: record for the §6.9 walk AND the §8.11.4 profiler
METHOD PROTECTED _M_SetStep
VAR_INPUT
    StepNo        : INT;
    StepName      : STRING(120);
    Awaits        : I_Module;
    AwaitingLabel : STRING(120);
    TimeClass     : E_TimeClass;
    ExpectedTime  : TIME;
END_VAR
VAR
    i : INT;
    e : ST_CondRecord;
END_VAR
IF StepNo <> CurrentStep.StepNo THEN
    _tStall(IN := FALSE);
    _M_ClearPending();
    FOR i := 1 TO PL_Fraktal.MAX_STEP_CONDS DO
        CurrentStep.Conds[i] := e;
    END_FOR
END_IF
CurrentStep.StepNo        := StepNo;
CurrentStep.StepName      := StepName;
CurrentStep.AwaitingLabel := AwaitingLabel;
CurrentStep.TimeClass     := TimeClass;
CurrentStep.ExpectedTime  := ExpectedTime;
_awaits := Awaits;
Profiler.StepChanged(StepNo := StepNo, StepName := StepName, TimeClass := TimeClass,
    Expected := ExpectedTime);
END_METHOD

// §6.9 — build the pending stall reason: step -> awaited command -> first FALSE condition
METHOD PROTECTED _M_StallWalk
IF Pending.ReasonCode = E_Reason.NONE THEN
    Pending.Since := F_Now();
END_IF
Pending.ReasonCode := E_Reason.STEP_STALLED;
Pending.Severity   := E_Severity.LOW;
Pending.Category   := E_Category.PROCESS;
Pending.SourcePath := _name;
Pending.Description := 'std.diagnostic.stepStalled';
END_METHOD

// §3.4.2 — the sequence author calls this at each step boundary; returns TRUE when
// the sequence may advance. Steppable (default TRUE) is the PER-STEP stop-point flag:
// a step with Steppable := FALSE runs straight through even in SINGLE_STEP/HOLD_TO_RUN
// (group several motions into one operator step, or a step unsafe to pause mid-way).
// CONTINUOUS: always TRUE. SINGLE_STEP: TRUE once per StepRequest edge (only if
// Steppable). HOLD_TO_RUN: TRUE while held (only if Steppable). Interlocks are
// enforced by the modules regardless (this only paces the sequence).
METHOD PROTECTED _M_StepGate : BOOL
VAR_INPUT
    Steppable : BOOL;
END_VAR
IF NOT Steppable THEN
    _M_StepGate := TRUE;               // not a stop point: advance regardless of run style
    RETURN;
END_IF
CASE RunStyle OF
    E_RunStyle.SINGLE_STEP:
        _stepArm(CLK := _stepReq);
        _stepReq := FALSE;
        _M_StepGate := _stepArm.Q;      // one advance per request edge
    E_RunStyle.HOLD_TO_RUN:
        _M_StepGate := _holdRun;        // advance only while held (NON-SAFETY)
ELSE
    _M_StepGate := TRUE;                // CONTINUOUS
END_CASE
END_METHOD

// §3.4 — override to declare the type's mode set (baseline: AUTO + MANUAL)
METHOD PROTECTED _M_Supports : BOOL
VAR_INPUT
    Mode : E_Mode;
END_VAR
_M_Supports := (Mode = E_Mode.AUTO) OR (Mode = E_Mode.MANUAL);
END_METHOD

// §3.4.2 — a concrete Unit overrides to opt a mode into SINGLE_STEP/HOLD_TO_RUN.
// Base: only CONTINUOUS.
METHOD PROTECTED _M_SupportsRunStyle : BOOL
VAR_INPUT
    Style : E_RunStyle;
END_VAR
_M_SupportsRunStyle := (Style = E_RunStyle.CONTINUOUS);
END_METHOD

// §6.11 — returns the chosen option once and clears the request (0 = none yet)
METHOD PROTECTED _M_TakeDecision : INT
IF DecisionAnswer > 0 THEN
    _M_TakeDecision := DecisionAnswer;
    DecisionAnswer := 0;
    Decision.Prompt := '';
ELSE
    _M_TakeDecision := 0;
END_IF
END_METHOD

// §8.11 — called by the chain/verdict glue at part completion
METHOD CountGood : BOOL
GoodCount := GoodCount + 1;
CountGood := TRUE;
END_METHOD

METHOD CountNok : BOOL
NokCount := NokCount + 1;
CountNok := TRUE;
END_METHOD

// §8.11.2 — REWORK verdict counter (see CountGood)
METHOD CountRework : BOOL
ReworkCount := ReworkCount + 1;
CountRework := TRUE;
END_METHOD

// §3.10.2 — Unit facets after the composite walk (own catalog + children):
// model catalog and per-mode switch policy, both static between config edits.
METHOD M_AppendConfig : BOOL
VAR_INPUT
    Pager : REFERENCE TO FB_ConfigPager;
END_VAR
VAR
    i    : INT;
    item : STRING(255);
END_VAR
M_AppendConfig := SUPER^.M_AppendConfig(Pager := Pager);
Pager.M_AppendNumber(Scope := Status.Name, Item := 'AvailableModelCount',
    Number := TO_DINT(AvailableModelCount));
FOR i := 1 TO AvailableModelCount DO
    item := CONCAT('AvailableModels/AvailableModels[',
        CONCAT(TO_STRING(i), ']/ModelCode'));
    Pager.M_Append(Scope := Status.Name, Item := item,
        ValueText := AvailableModels[i].ModelCode);
END_FOR
FOR i := 0 TO PL_Fraktal.MODE_COUNT - 1 DO
    item := CONCAT('ModePolicy/ModePolicy[', CONCAT(TO_STRING(i), ']/Shield'));
    Pager.M_AppendNumber(Scope := Status.Name, Item := item,
        Number := TO_DINT(ModePolicy[i].Shield));
    item := CONCAT('ModePolicy/ModePolicy[', CONCAT(TO_STRING(i), ']/Style'));
    Pager.M_AppendNumber(Scope := Status.Name, Item := item,
        Number := TO_DINT(ModePolicy[i].Style));
END_FOR
END_METHOD

METHOD M_SequenceAskDecision
VAR_INPUT
    Req : ST_DecisionRequest;
END_VAR
_M_AskDecision(Req := Req);
END_METHOD

METHOD M_SequenceAwait : BOOL
VAR_INPUT
    Idx : INT;
    Label : STRING(120);
    Ok : BOOL;
END_VAR
M_SequenceAwait := _M_Await(Idx := Idx, Label := Label, Ok := Ok);
END_METHOD

METHOD M_SequenceClearDecision
Decision.Prompt := '';
DecisionAnswer := 0;
END_METHOD

METHOD M_SequenceComplete
_M_Complete();
END_METHOD

METHOD M_SequenceCountGood
CountGood();
END_METHOD

METHOD M_SequenceEndOfCycle : BOOL
M_SequenceEndOfCycle := _M_EndOfCycle();
END_METHOD

METHOD M_SequenceFault
VAR_INPUT
    Reason : E_Reason;
    DescriptionKey : STRING(255);
END_VAR
_M_Fault(Reason, DescriptionKey);
END_METHOD

METHOD M_SequencePartProcessed : BOOL
VAR_INPUT
    Verdict : E_Verdict;
    Reason : E_Reason;
END_VAR
M_SequencePartProcessed :=
    _M_PartProcessed(Verdict := Verdict, Reason := Reason);
END_METHOD

METHOD M_SequencePartReceived : BOOL
M_SequencePartReceived := _M_PartReceived();
END_METHOD

METHOD M_SequencePartRecord : BOOL
VAR_INPUT
    RecordName : STRING(64);
    Value : LREAL;
    Minimum : LREAL;
    Maximum : LREAL;
    Target : LREAL;
    EngUnit : STRING(16);
END_VAR
M_SequencePartRecord := _M_PartRecord(RecordName := RecordName,
    Value := Value, Minimum := Minimum, Maximum := Maximum, Target := Target,
    EngUnit := EngUnit);
END_METHOD

METHOD M_SequencePartStarted
_M_PartStarted();
END_METHOD

// I_SequenceHost (§6.7/§6.8) — step record for a separately-compiled chain.
METHOD M_SequenceSetStep
VAR_INPUT
    StepNo : INT;
    StepName : STRING(120);
    Awaits : I_Module;
    AwaitingLabel : STRING(120);
    TimeClass : E_TimeClass;
    ExpectedTime : TIME;
END_VAR
_M_SetStep(StepNo := StepNo, StepName := StepName,
    Awaits := Awaits, AwaitingLabel := AwaitingLabel, TimeClass := TimeClass,
    ExpectedTime := ExpectedTime);
END_METHOD

METHOD M_SequenceStepGate : BOOL
VAR_INPUT
    Steppable : BOOL;
END_VAR
M_SequenceStepGate := _M_StepGate(Steppable := Steppable);
END_METHOD

// §3.4/§8.11 — accept a pending Stop BETWEEN cycles: the open profile fragment
// (just the wait step) is abandoned, not published as a production cycle.
METHOD M_SequenceStopNow
Profiler.CycleAbandon();
_stopReq := FALSE;
Execute := FALSE;
_M_Complete();
END_METHOD

// §3.4 — a chain polls this at its between-cycles wait step.
METHOD M_SequenceStopPending : BOOL
M_SequenceStopPending := _stopReq AND (_exec = E_ExecState.BUSY);
END_METHOD

METHOD M_SequenceTakeDecision : INT
M_SequenceTakeDecision := _M_TakeDecision();
END_METHOD

// §7.6.1 — single gated manual-command entry for the HMI. Accepts ONLY when this
// Unit is in MANUAL (§3.4) AND the user holds MANUAL access (§7.7). Routes to the
// target module's ManualCommand (through the command surface — defended, not
// bypassed). Logs every accept/reject as a §8.3 event. Concrete Units override
// _M_RouteManual to map TargetPath -> the child module.
METHOD ManualCommandTo : BOOL
VAR_INPUT
    TargetPath : STRING(255);
    Value : DINT;
END_VAR
VAR
    auditSlot : INT;
END_VAR
ManualCommandTo := FALSE;
IF _mode <> E_Mode.MANUAL THEN
    auditSlot := AlarmLog.Raise(Reason := E_Reason.NONE,
        Text := 'std.audit.manualCommandWrongMode', Source := TargetPath,
        Severity := E_Severity.LOW, Category := E_Category.SYSTEM, ResetClass := E_ResetClass.AUTO_RESET);
    IF auditSlot > 0 THEN AlarmLog.Gone(Slot := auditSlot); END_IF
    RETURN;
END_IF
IF NOT Access.PermitsLogged(Gate := E_GatedAction.MANUAL) THEN
    RETURN;                              // §7.7 denial already audited
END_IF
ManualCommandTo := _M_RouteManual(TargetPath := TargetPath, Value := Value);
IF ManualCommandTo THEN
    auditSlot := AlarmLog.Raise(Reason := E_Reason.NONE,
        Text := 'std.audit.manualCommandAccepted', Source := TargetPath,
        Severity := E_Severity.LOW, Category := E_Category.SYSTEM, ResetClass := E_ResetClass.AUTO_RESET);
ELSE
    auditSlot := AlarmLog.Raise(Reason := E_Reason.UNSUPPORTED_COMMAND,
        Text := 'std.audit.manualCommandRejected', Source := TargetPath,
        Severity := E_Severity.LOW, Category := E_Category.SYSTEM, ResetClass := E_ResetClass.AUTO_RESET);
END_IF
IF auditSlot > 0 THEN AlarmLog.Gone(Slot := auditSlot); END_IF
END_METHOD

PROPERTY ModeActive : E_Mode
GET
ModeActive := _mode;
END_GET
END_PROPERTY

PROPERTY ModelCode : STRING(64)
GET
ModelCode := Model.ModelCode;
END_GET
END_PROPERTY

PROPERTY ModuleType : E_ModuleType
GET
ModuleType := E_ModuleType.UNIT;
END_GET
END_PROPERTY

